	//定位状态更新
	//定位完成状态
	IF (iPosId<>-1) AND (bPosDone1 OR bPosDone2) THEN									                                             
	 		bGo_OK := TRUE;
			stAxis.Pos.State.bGo_Moving:=FALSE;		
			iPosId:=-1;
	END_IF;
	//定位完成与位置共同判断	 
	IF	 bRelEx THEN			 
		stAxis.Pos.State.bGo_OK	:=  bGo_OK (*AND (ABS((rPosEx + rRelStartPos)- stAxis.State.rActPos )<= stAxis.Parameter.rInPosValue)*);
	ELSE	
		stAxis.Pos.State.bGo_OK	:=  bGo_OK AND (ABS(stAxis.Pos.Par.rPos - stAxis.State.rActPos )<= stAxis.Parameter.rInPosValue);
	END_IF
		 
	//定位中状态
	IF (bPosBusy1 OR bPosBusy2)  THEN																						
	 	bGo_OK := FALSE;
		stAxis.Pos.State.bGo_Moving:=TRUE;				
	END_IF;
	//未定位中，清空定位ID号
	IF NOT bPosBusy1 AND NOT bPosBusy2 THEN  																
		iPosId:=-1;
	END_IF;
	
	//定位计时
	TonAxisMove(IN:=(iPosId <> -1), PT:= T#9999S);
	IF iPosId <> -1 THEN
		stAxis.Pos.State.rGo_CT:=TIME_TO_REAL(TonAxisMove.ET)/1000.0;	
	END_IF;	
END_IF;
{endregion}
END_ACTION

ACTION A_09_Stop:
{region "轴停止"}
IF TRUE THEN
	IF bHoming THEN
		lrStopMoveDec:=stAxis.Parameter.rStopDec * 1000.0;
	ELSE
		lrStopMoveDec:=stAxis.Parameter.rStopDec * 1000.0;
	END_IF;
		
	bStopMoveExe:= (stAxis.Control.bStop_M AND stSystem.bManual) OR stAxis.Control.bStop_A OR stSystem.bStop;
	IF bStopMoveExe (*AND NOT bStopMoveExeLast *)THEN
		bHomeJogBExe := FALSE ;
		bHomeJogFExe := FALSE ;	
		bHoming:= FALSE;
		iHomeStep:=0;
		iHomeStepPre := 0;
		stAxis.Pos.State.bGo_Moving:=FALSE;
		iPosId:=-1;
//		uiMotionCMD:=5;
	END_IF;
	bStopExe:= bHomeStop OR bStopMoveExe OR stAxis.State.bError OR stSystem.bEMG ;
	fbMcStop(
		Axis:= AxisRef, 
		Execute:= bStopExe  , 
		Deceleration:= lrStopMoveDec , 
		Jerk:= lrStopMoveDec * REAL#10.0	 , 
		Options:= , 
		Done=> , 
		Busy=> , 
		Active=> , 
		CommandAborted=> , 
		Error=> , 
		ErrorID=> );
	
	bHomeStop:=FALSE;
	IF stAxis.State.bStandStill AND ((stAxis.Control.bStop_M AND stSystem.bManual) OR stAxis.Control.bStop_A) THEN
		stAxis.Control.bStop_A:=FALSE;
		stAxis.Control.bStop_M:=FALSE;
	END_IF;
	bStopMoveExeLast:=bStopMoveExe;
END_IF;
{endregion}
END_ACTION

ACTION A_10_TrqCtr:
{region "力矩切换"}

// 转矩模式下，力矩切换
// 转矩6071目标转矩的单位为 0.1% ，上位机按照百分比输出，数据转换 *10

iTorqueTemp := REAL_TO_INT(stAxis.Parameter.rTorque *10)	;
	 
IF stAxis.State.siModeOfOperation = 10 THEN	// 驱动器处于转接模式时可设定力矩
	fbEcCoeSdoWriteExTargetTrq(
	sNetId:=strDriveAddressNetID , 
	nSlaveAddr:= uiDriveAddressSlaveAddr, 
	nSubIndex:= 16#00, 
	nIndex:= (16#6071 + (stAxis.Parameter.uiAxisChannelNum - 1)*16#800), 
	pSrcBuf:= ADR(iTorqueTemp), 
	cbBufLen:= SIZEOF(iTorqueTemp), 
	bExecute:= iTorqueTemp<> iTorqueTempOld , 
	tTimeout:= , 
	bCompleteAccess:= , 
	bBusy=> , 
	bError=> , 
	nErrId=> );	 
END_IF
iTorqueTempOld := iTorqueTemp;
	 
{endregion}
END_ACTION

ACTION A_11_StateOut:
{region "状态输出"}
//绝对值编码器电机在驱动器中设置好原点，默认原点OK
//增量式编码器需程序回零
IF  stAxis.Parameter.bAbsEnc AND stAxis.Control.bHome_A THEN
	stAxis.State.bHome_OK := TRUE;
	stAxis.Control.bHome_A:=FALSE;
ELSE
	stAxis.State.bHome_OK :=(AxisRef.Status.Homed OR stAxis.State.bHome_OK)
							AND NOT AxisRef.Status.DriveDeviceError;
	stAxis.State.bHoming :=(AxisRef.Status.Homing OR bHoming)
							AND NOT AxisRef.Status.DriveDeviceError;
END_IF;

//模轴和线性轴当前位置输出
stAxis.State.rActModuloPos := LREAL_TO_REAL(AxisRef.NcToPlc.ModuloActPos);
stAxis.State.rActPos := LREAL_TO_REAL(AxisRef.NcToPlc.ActPos);
//速度转矩加速度
stAxis.State.rActVel :=LREAL_TO_REAL(AxisRef.NcToPlc.ActVelo);
stAxis.State.rActTrq :=LREAL_TO_REAL(AxisRef.NcToPlc.ActTorque);
stAxis.State.rActAcc :=LREAL_TO_REAL(AxisRef.NcToPlc.ActAcc);
{endregion}
END_ACTION

ACTION A_12_Error:
{region "轴报警"}
//报警复位
IF ((stSystem.bReset OR stAxis.Control.bReset_A OR (stAxis.Control.bReset_M AND stSystem.bManual)) AND NOT bResetLast ) THEN
	FOR m:=1 TO 12 BY 1 DO
		stAxis.state.arErrorID[m]:= FALSE;
	END_FOR;
	stAxis.State.bWarning := FALSE;
	stAxis.State.bLightEror := FALSE;
	stAxis.State.bCriticalError :=FALSE;
END_IF;
bResetLast := stSystem.bReset;

//轴报警1-轴未使能
//屏蔽轴未使能报警
RtrigPowerOn(CLK:=stAxis.State.bPowerOK , Q=> );
//bHoming状态在驱动器回零时使用
IF NOT stAxis.State.bPowerOK AND NOT bHoming AND FALSE THEN
	stAxis.State.bLightEror := TRUE;
	stAxis.State.arErrorID[1]:=TRUE;
END_IF;
(*
IF RtrigPowerOn.Q THEN
	stAxis.State.bLightEror:=FALSE;
	stAxis.State.arErrorID[0]:=FALSE;
	stAxis.State.wstrErrorInfo:="--";
END_IF;
*)
	 
//轴报警2-轴NC报警
IF AxisRef.Status.ErrorID > 0 AND (NOT mcReset.Busy AND (NOT bHoming (*AND stAxis.Parameter.uiHomeMode <>6*))) THEN
	stAxis.State.bCriticalError := TRUE;
	stAxis.State.arErrorID[2]:=TRUE;
END_IF;
		  
//轴报警3-驱动器报警
TonReadDriveErrorCode(IN:=AxisRef.Status.DriveDeviceError,PT:=TIME#50MS);
IF AxisRef.Status.DriveDeviceError AND NOT mcReset.Busy AND TonReadDriveErrorCode.Q THEN
	stAxis.State.bCriticalError := TRUE;
	stAxis.State.arErrorID[3]:=TRUE;
END_IF;	 	 

//轴报警4-回零条件不满足报警
IF stAxis.Control.bHome_A AND NOT stAxis.Control.bHome_Con THEN
	stAxis.State.bLightEror := TRUE;
	stAxis.State.arErrorID[4]:=TRUE;
END_IF;	 

//轴报警5-正向JOG运行条件不满足报警
IF((stAxis.Control.bJogCw_A OR (stAxis.Control.bJogCw_M AND stSystem.bManual))AND NOT stAxis.Control.bJogCw_Con) THEN 
	stAxis.State.bLightEror := TRUE;
	stAxis.State.arErrorID[5]:=TRUE;
END_IF;

//轴报警6-负向JOG运行条件不满足报警
IF( (stAxis.Control.bJogCcw_A OR (stAxis.Control.bJogCcw_M AND stSystem.bManual)) AND NOT stAxis.Control.bJogCcw_Con) THEN 
	stAxis.State.bLightEror := TRUE;
	stAxis.State.arErrorID[6]:=TRUE;
END_IF;

//轴报警7-运行方向错误报警
IF ((stAxis.State.bPsw AND bHomeJogFExe) OR (stAxis.State.bNSw AND bHomeJogBExe)) AND NOT (stAxis.Parameter.uiHomeMode = 6 AND iHomeStepPre > 0 AND iHomeStep<1000) THEN
	bHomeJogFExe := FALSE;
	bHomeJogbExe := FALSE;
	bWrongDirection := TRUE;
END_IF;
IF stSystem.bReset OR stAxis.Control.bReset_A OR (stAxis.Control.bReset_M AND stSystem.bManual) THEN
	bWrongDirection := FALSE;
END_IF;
IF bWrongDirection THEN
	stAxis.State.bLightEror :=TRUE;
	stAxis.State.arErrorID[7]:=TRUE;
END_IF;
	 		   
//轴报警8-运行中碰正限位报警
RtrigJogB(CLK:=bJogBExe , Q=> );
IF (NOT stAxis.State.bPSw AND stAxis.State.bDirPositive ) AND NOT bHoming THEN 
	stAxis.State.bCriticalError :=TRUE;
	stAxis.State.arErrorID[8]:=TRUE;
END_IF;
IF RtrigJogB.Q AND stAxis.State.bPSw THEN
	stAxis.State.bCriticalError :=FALSE;
	stAxis.State.arErrorID[8]:=FALSE;
END_IF

// 轴报警9-运行中碰负限位报警
RtrigJogF(CLK:=bJogFExe , Q=> );
IF (NOT stAxis.State.bNSw AND stAxis.State.bDirNegative ) AND NOT bHoming THEN 
	stAxis.State.bCriticalError :=TRUE;
	stAxis.State.arErrorID[9]:=TRUE;
END_IF;
IF RtrigJogF.Q AND stAxis.State.bNSw THEN
	stAxis.State.bCriticalError :=FALSE;
	stAxis.State.arErrorID[9]:=FALSE;
END_IF

//
stAxis.state.bError := stAxis.State.bCriticalError OR stAxis.State.bLightEror ;
{endregion}


//报警输出	 
{region "SetAlarm"}
//SetAlarm
//轴报警从编号 101 开始, 12 个为一组
arrfbSetAlarm[1](
	bEnable:= TRUE, 
	iErrorID:= 100 + (UDINT_TO_INT(AxisREF.NcToPlc.AxisId)-1) * 12 + 1, 
	bExecute:= stAxis.State.arErrorID[1], 
	bReset:= stSystem.bReset OR stAxis.Control.bReset_A OR (stAxis.Control.bReset_M AND stSystem.bManual), 
	strErrorInfoEN:= 'not enabled', 
	wstrErrorInfoCN:= "轴未使能", 
	enumErrorClass:= 6, 
	 );
arrfbSetAlarm[2](
	bEnable:= TRUE, 
	iErrorID:= 100 + (UDINT_TO_INT(AxisREF.NcToPlc.AxisId)-1) * 12 + 2, 
	bExecute:= stAxis.State.arErrorID[2], 
	bReset:= stSystem.bReset OR stAxis.Control.bReset_A OR (stAxis.Control.bReset_M AND stSystem.bManual), 
	strErrorInfoEN:= 'NC alarm', 
	wstrErrorInfoCN:= "轴NC报警,报警代码-", 
	enumErrorClass:= 7,
	wstr1:=STRING_TO_WSTRING(stAxis.strName),
	D1:=UDINT_TO_DINT(AxisRef.Status.ErrorID),
	 );
arrfbSetAlarm[3](
	bEnable:= TRUE, 
	iErrorID:= 100+ (UDINT_TO_INT(AxisREF.NcToPlc.AxisId)-1) * 12 + 3, 
	bExecute:= stAxis.State.arErrorID[3], 
	bReset:= stSystem.bReset OR stAxis.Control.bReset_A OR (stAxis.Control.bReset_M AND stSystem.bManual), 
	strErrorInfoEN:= 'drive alarm', 
	wstrErrorInfoCN:= "驱动器报警,报警代码-", 
	enumErrorClass:= 7,
	wstr1:=STRING_TO_WSTRING(stAxis.strName),
	D1:=UDINT_TO_DINT(stAxis.State.uiDriveErrorCode),
	 );
arrfbSetAlarm[4](
	bEnable:= TRUE, 
	iErrorID:= 100+ (UDINT_TO_INT(AxisREF.NcToPlc.AxisId)-1) * 12 + 4, 
	bExecute:= stAxis.State.arErrorID[4], 
	bReset:= stSystem.bReset OR stAxis.Control.bReset_A OR (stAxis.Control.bReset_M AND stSystem.bManual), 
	strErrorInfoEN:= 'home condition not satisfied', 
	wstrErrorInfoCN:= "回零条件不满足", 
	wstr1:=STRING_TO_WSTRING(stAxis.strName),
	enumErrorClass:= 6, 
	 );	
arrfbSetAlarm[5](
	bEnable:= TRUE, 
	iErrorID:= 100+ (UDINT_TO_INT(AxisREF.NcToPlc.AxisId)-1) * 12 + 5, 
	bExecute:= stAxis.State.arErrorID[5], 
	bReset:= stSystem.bReset OR stAxis.Control.bReset_A OR (stAxis.Control.bReset_M AND stSystem.bManual), 
	strErrorInfoEN:= 'positive JOG condition not satisfied', 
	wstrErrorInfoCN:= "正向JOG运行条件不满足", 
	wstr1:=STRING_TO_WSTRING(stAxis.strName),
	enumErrorClass:= 6, 
	 );	 
arrfbSetAlarm[6](
	bEnable:= TRUE, 
	iErrorID:= 100+ (UDINT_TO_INT(AxisREF.NcToPlc.AxisId)-1) * 12 + 6, 
	bExecute:= stAxis.State.arErrorID[6], 
	bReset:= stSystem.bReset OR stAxis.Control.bReset_A OR (stAxis.Control.bReset_M AND stSystem.bManual), 
	strErrorInfoEN:= 'negative JOG condition not satisfied', 
	wstrErrorInfoCN:= "反向JOG运行条件不满足", 
	wstr1:=STRING_TO_WSTRING(stAxis.strName),
	enumErrorClass:= 6, 
	 );	 
arrfbSetAlarm[7](
	bEnable:= TRUE, 
	iErrorID:= 100+ (UDINT_TO_INT(AxisREF.NcToPlc.AxisId)-1) * 12 + 7, 
	bExecute:= stAxis.State.arErrorID[7], 
	bReset:= stSystem.bReset OR stAxis.Control.bReset_A OR (stAxis.Control.bReset_M AND stSystem.bManual), 
	strErrorInfoEN:= 'wrong direction of motion', 
	wstrErrorInfoCN:= "回零过程中JOG运行方向错误", 
	wstr1:=STRING_TO_WSTRING(stAxis.strName),
	enumErrorClass:= 6, 
	 );
arrfbSetAlarm[8](
	bEnable:= TRUE, 
	iErrorID:= 100+ (UDINT_TO_INT(AxisREF.NcToPlc.AxisId)-1) * 12 + 8, 
	bExecute:= stAxis.State.arErrorID[8], 
	bReset:= stSystem.bReset OR stAxis.Control.bReset_A OR (stAxis.Control.bReset_M AND stSystem.bManual), 
	strErrorInfoEN:= 'positive limit alarm', 
	wstrErrorInfoCN:=  "正限位报警", 
	wstr1:=STRING_TO_WSTRING(stAxis.strName),
	enumErrorClass:= 6, 
	 );
arrfbSetAlarm[9](
	bEnable:= TRUE, 
	iErrorID:= 100+ (UDINT_TO_INT(AxisREF.NcToPlc.AxisId)-1) * 12 + 9 , 
	bExecute:= stAxis.State.arErrorID[9], 
	bReset:= stSystem.bReset OR stAxis.Control.bReset_A OR (stAxis.Control.bReset_M AND stSystem.bManual), 
	strErrorInfoEN:= 'negative limit alarm', 
	wstrErrorInfoCN:=  "负限位报警",
	wstr1:=STRING_TO_WSTRING(stAxis.strName), 
	enumErrorClass:= 6, 
	 );		  
//轴报警10
arrfbSetAlarm[10](
	bEnable:= TRUE, 
	iErrorID:= 100+ (UDINT_TO_INT(AxisREF.NcToPlc.AxisId)-1) * 12 + 10, 
	bExecute:= stAxis.State.arErrorID[10], 
	bReset:= stSystem.bReset OR stAxis.Control.bReset_A OR (stAxis.Control.bReset_M AND stSystem.bManual), 
	strErrorInfoEN:= 'homing process interruption,step:', 
	wstrErrorInfoCN:=  "回零流程异常，步序-",	
	enumErrorClass:= 6, 
	wstr1:=STRING_TO_WSTRING(stAxis.strName),
	D1:=INT_TO_DINT(iHomeStep),
	 );

//轴报警11
arrfbSetAlarm[11](
	bEnable:= TRUE, 
	iErrorID:= 100 + (UDINT_TO_INT(AxisREF.NcToPlc.AxisId)-1) * 12 + 11, 
	bExecute:= stAxis.State.arErrorID[11], 
	bReset:= stSystem.bReset OR stAxis.Control.bReset_A OR (stAxis.Control.bReset_M AND stSystem.bManual), 
	strErrorInfoEN:= 'Positioning motion conditions are not met.', 
	wstrErrorInfoCN:=  "定位运动条件不满足", 
	wstr1:=STRING_TO_WSTRING(stAxis.strName),
	enumErrorClass:= 6, 
	 );
//轴报警12
arrfbSetAlarm[12](
	bEnable:= TRUE, 
	iErrorID:= 100 + (UDINT_TO_INT(AxisREF.NcToPlc.AxisId)-1) * 12 + 12, 
	bExecute:= stAxis.State.arErrorID[12], 
	bReset:= stSystem.bReset OR stAxis.Control.bReset_A OR (stAxis.Control.bReset_M AND stSystem.bManual), 
	strErrorInfoEN:= 'Positioning conditions not met during motion', 
	wstrErrorInfoCN:=  "运动中定位条件不满足", 
	wstr1:=STRING_TO_WSTRING(stAxis.strName),
	enumErrorClass:= 6, 
	 );
{endregion}
END_ACTION

END_FUNCTION_BLOCK

// ---- FB/61_Alarm/FB/FB_SetError.TcPOU
FUNCTION_BLOCK FB_SetError
VAR_INPUT
	//是否启用当前报警
    bEnable						:                   BOOL						;
	//当前报警的报警代码号
	iErrorID					:					INT							;
	//当前报警的触发信号输入
	bExecute						:					BOOL						;
END_VAR
VAR_INPUT
	//报警复位信号输入
	bReset						:					BOOL						;
	// 报警信息-英文字符
	strErrorInfoEN				: 					STRING						;
	// 报警信息-中文字符
	wstrErrorInfoCN				: 					WSTRING						;
	//当前报警的等级设定
	enumErrorClass				:					Enum_ErrorClass				;
END_VAR
VAR_INPUT
	//报警发生时，需要触发的动作，1-4中任意选择。                           						
	bAlarmAction1				:					BOOL						;
	bAlarmAction2				:					BOOL						;
	bAlarmAction3				:					BOOL						;
	bAlarmAction4				:					BOOL						;
	// 报警代码的对应轴名称，驱动器报警时可以调用
	wstr1						: 					WSTRING						;
	// 报警代码，NC报警代码，驱动器报警代码
	D1							:					DINT						;
END_VAR
VAR_OUTPUT
	// 报警启用标志位
	bEnabled					: 					BOOL						;
	// 报警发生标志位
	bErrorOccur					:					BOOL						;
END_VAR
VAR
	(**暂时不启用，需要时添加至输入变量中**)
	//是否对当前报警启用滤波功能(**暂时不启用，需要时添加至输入变量中**)
   bFilterOn					:                  	BOOL:=FALSE					;
	//滤波功能的时间设定(**暂时不启用，需要时添加至输入变量中**)
   timeFilter					:                   TIME := TIME#0MS			;	
	// 是否使用reset信号复位:  true=复位信号为1时且触发信号为0时，复位报警状态;  false=触发信号为0时自动复位报警信号(**暂时不启用，需要时添加至输入变量中**)
	bResetSignalUse				:					BOOL := TRUE				;	
	//设定是否将当前报警记录到历史记录中(**暂时不启用，需要时添加至输入变量中**)
   	bSavetoHistory				:                 	BOOL := TRUE				;
	strVersion: STRING;

	
	// 获取报警时间
	rtrigGetTime				:          			R_TRIG						;
  	// 滤波延时
	tonFilter					:               	TON							;	
 	// 报警复位信号下降沿
	ftrigResetExe				:          			F_TRIG						;	
	i							:                 	INT							;
	strTemp						: 					STRING						;
	fbFormatStringDateTime		: 					FB_FormatString				;
	strDateTime					: 					STRING(255)					;
	wstrErrorMessage			: 					WSTRING						;
	bFirstRun: BOOL := true;
	ton100msDelay: TON;
END_VAR

(***
by Yu
	
	2025-07-23	报警设置功能块，每一个报警都需实例化一次。
	2025-07-24	输出的报警信息中不同时整合报警时间和报警ID号,减少字符的使用长度。报警时间、报警ID号、报警信息，以结构体的形式分别输出。
	2025-10-29	报警发生时，增加获取系统时间判定，防止出现开机一瞬间，系统时间还未获取时，出现的错误时间报警


***)
//当前版本更新时间
strVersion := '2025-10-29' ;

//初始化
IF bFirstRun THEN
;
END_IF


//报警ID号超范围直接退出
IF iErrorID> iErrorIDMax OR iErrorID< 1 THEN
	RETURN;
END_IF

//报警复位
 ftrigResetExe(CLK:=bReset);
 IF ((bResetSignalUse AND  ftrigResetExe.Q)OR NOT bResetSignalUse )AND NOT bExecute OR NOT bEnable THEN
    bErrorOccur:=FALSE;
    arrstError[iErrorID].bAlarmAction1:=FALSE;
    arrstError[iErrorID].bAlarmAction2:=FALSE;
    arrstError[iErrorID].bAlarmAction3:=FALSE;
    arrstError[iErrorID].bAlarmAction4:=FALSE;
	arrstError[iErrorID].bEnabled:=bEnable;
	arrstError[iErrorID].bErrorOccur:=bErrorOccur;
	arrstError[iErrorID].bErrorExe:=bExecute;
	arrstError[iErrorID].enumErrorClass:=enumErrorClass;
	arrstError[iErrorID].iErrorID:=iErrorID;
	arrstError[iErrorID].bResetExe:=bReset;
	arrstError[iErrorID].bResetSignalUse:=bResetSignalUse;
 END_IF
 
	
//滤波延时
tonFilter(IN:=bFilterOn AND bExecute , PT:=timeFilter );

//报警发生上升沿触发且系统时间读取成功
rtrigGetTime(CLK:=((NOT bFilterOn ) OR (bFilterOn AND tonFilter.Q))AND bEnable AND bExecute AND bGetSystemTimeDone  );

//将当前系统时间写入到对应的轴结构体中 
IF rtrigGetTime.Q THEN
	arrstError[iErrorID].dtErrorOccorTime:=SYSTEMTIME_TO_DT(tActSystemTime);
END_IF

//报警发生时触发
IF ((NOT bFilterOn ) OR (bFilterOn AND tonFilter.Q)) AND bEnable AND bExecute AND bGetSystemTimeDone THEN
	//报警发生标志位
	bErrorOccur:=TRUE;
	//将报警后的触发动作写入对应的ErrorID号下
	arrstError[iErrorID].bAlarmAction1:=bAlarmAction1;
	arrstError[iErrorID].bAlarmAction2:=bAlarmAction2;
	arrstError[iErrorID].bAlarmAction3:=bAlarmAction3;
	arrstError[iErrorID].bAlarmAction4:=bAlarmAction4;
	//设定此ErrorID号报警是否启用
	arrstError[iErrorID].bEnabled:=bEnable;
	//此ErrorID号报警发生标志位
	arrstError[iErrorID].bErrorOccur:=bErrorOccur;
	//此ErrorID号报警触发信号
	arrstError[iErrorID].bErrorExe:=bExecute;
	//此ErrorID号报警警报等级	
	arrstError[iErrorID].enumErrorClass:=enumErrorClass;
	//此ErrorID号报警报警ID	
	arrstError[iErrorID].iErrorID:=iErrorID;
	//此ErrorID号报警报警复位信号		
	arrstError[iErrorID].bResetExe:=bReset;
	//设定此ErrorID号报警是否与复位信号联动
	arrstError[iErrorID].bResetSignalUse:=bResetSignalUse;
END_IF

//报警发生时的时间转换程string类型。时间-报警ID号-报警信息，组合输出
IF rtrigGetTime.Q THEN
	fbFormatStringDateTime(
		sFormat:= '%D-%D-%D-%D:%D:%D',
		arg1:= F_WORD(tActSystemTime.wYear),
		arg2:= F_WORD(tActSystemTime.wMonth),
		arg3:= F_WORD(tActSystemTime.wDay),
		arg4:= F_WORD(tActSystemTime.wHour),
		arg5:= F_WORD(tActSystemTime.wMinute),
		arg6:= F_WORD(tActSystemTime.wSecond),
		sOut=> strDateTime
		);
	//默认使用中文报警信息
	IF bLanguageSet=1 THEN
		wstrErrorMessage:=STRING_TO_WSTRING(strErrorInfoEN);
	ELSE
		wstrErrorMessage:=wstrErrorInfoCN;
	END_IF	
	F_FormatWstringErrInfo(wstrIn:=wstrErrorMessage,wstrPreMessage:=wstr1,diMessage:=D1,wstrOut=>wstrErrorMessage);	
	//整合需要添加的字符后，直接输出，不添加报警时间以及报警ID，减少字符的长度
	arrstError[iErrorID].wstrErrorMessage := wstrErrorMessage ;	
//	wstrErrorMessage:=	WCONCAT(WCONCAT(WCONCAT("ID",INT_TO_WSTRING(iErrorID)),","),wstrErrorMessage);		
//	arrstError[iErrorID].wstrErrorMessage := WCONCAT(WCONCAT(STRING_TO_WSTRING(strDateTime),"-"),wstrErrorMessage);	
END_IF
	   

//当选择将此报警记录如历史报警记录后，触发记录。最大记录数组200组。数据向后依次排列
IF bSavetoHistory  AND rtrigGetTime.Q THEN
	iHistoryErrorNum:=iHistoryErrorNum+1;
	IF iHistoryErrorNum>=200 THEN
		iHistoryErrorNum:=200;
	END_IF
	IF iHistoryErrorNum>=2 THEN
		FOR i:=iHistoryErrorNum TO 2 BY -1 DO
			arrstHistoryError[i]:=arrstHistoryError[i-1];
		END_FOR
	END_IF
 	arrstHistoryError[1].iErrorID:=iErrorID;
	arrstHistoryError[1].dtErrorTime:=arrstError[iErrorID].dtErrorOccorTime;
  	arrstHistoryError[1].wstrErrorMessage:=arrstError[iErrorID].wstrErrorMessage;
END_IF

END_FUNCTION_BLOCK

// ---- FB/61_Alarm/FB/F_FormatWstringErrInfo.TcPOU
FUNCTION F_FormatWstringErrInfo : WSTRING
FUNCTION F_FormatWstringErrInfo : BOOL
VAR_INPUT
	wstrIn:			WSTRING;
	// 前缀
	wstrPreMessage: WSTRING;
	// 后缀
	diMessage:					DINT;
END_VAR
VAR_OUTPUT
	wstrOut:			WSTRING;
END_VAR
VAR
	strVersion: STRING;
	iVar0: INT;
	iVar1: INT;
	iVar2: DINT;
	wstrTemp: WSTRING;
END_VAR

(***
by Yu
	
	2025-07-23	实现对信息的组合,前缀为 WSTRING 变量，后缀添加 DINT 型变量。可用于添加 轴名称-报警信息-报警代码 。

***)
//当前版本更新时间
strVersion := '2025-07-23' ;

//
iVar0:=WLEN(wstrIn);
iVar1:=WLEN(wstrPreMessage);
iVar2:=diMessage;

IF iVar1 <>0 AND iVar2 <>0 THEN
	wstrTemp := WCONCAT(wstrPreMessage,wstrIn);
	wstrOut := WCONCAT(wstrtemp,DINT_TO_WSTRING(diMessage));
ELSIF iVar1 = 0 AND iVar2 <> 0  THEN
	wstrOut := WCONCAT(wstrIn,DINT_TO_WSTRING(diMessage));
ELSIF iVar1 <>0 AND iVar2 =0 THEN
	wstrOut := WCONCAT(wstrPreMessage,wstrIn);	
ELSE
	wstrOut := wstrIn;
END_IF

END_FUNCTION

// ---- FB/01_Axis/FB/FB_TouchProbe_Home_Bylimit.TcPOU
FUNCTION_BLOCK FB_TouchProbe_Home_Bylimit
VAR_INPUT	
		bCMD_HomeExecute			:REFERENCE TO BOOL;			(* 执行回零*)
		bCMD_Reset					:REFERENCE TO BOOL;			(* 回零错误复位*)
		bCMD_EnableState			:BOOL;						(* 使能状态输入*)	
		bCMD_StartHomeIndex			:BOOL;						(* 是否使用索引回零*)
		eCMD_HomeDirection			:MC_Direction;				(* 回原点方向*)
		bCMD_PositiveLimit			:BOOL;						(* 正限位传感器*)
		bCMD_NegativeLimit			:BOOL;						(* 负限位传感器*)
		rCMD_HomePosition			:LREAL;						(* 设定回原点位置*)
		rCMD_TowardsVelSetValue		:LREAL;						(* 靠近原点速度*)
		rCMD_OffVelSetValue			:LREAL;						(* 离开原点速度*)
	    stHomeAdsGroup				:ST_HomeAdsGroup;			(* ADS地址信息*)

END_VAR
VAR_OUTPUT
		bResult_HomeDone			:BOOL;						(* 回原点完成状态*)
		bResult_HomeBusy			:BOOL;						(* 正在回原点中状态*)
		bResult_HomeError			:BOOL;						(* 回原点错误状态*)
		nResult_HomeErrorID			:UDINT;						(* 回原点错误代码*)
END_VAR
VAR_IN_OUT
		axis						:AXIS_REF;
END_VAR
VAR
	  
		mcHome						:MC_Home;
		mcReset						:MC_Reset;
		fbReadParameter				:ARRAY [0..4] OF ADSREAD;
		fbwriteParameter			:ARRAY [0..4] OF ADSWRITE;
		rTowardsVelActValue			:LREAL;		
		rOffVelActValue				:LREAL;
		nHomeSenorSetValue			:INT;
		nHomeSensorActValue			:INT;
		nHomeSynSetValue			:WORD;
		nHomeSynActValue			:WORD;
		nHomeSetRefMode				:DINT;
		nHomeActRefMode				:DINT;
		mcHomeStatus				:ST_McOutputs;
		fbReadParaStatus			:ARRAY [0..4] OF ST_McOutputs;
		fbWriteParaStatus			:ARRAY [0..4] OF ST_McOutputs;
		posEdge_bCMD_HomeExecute	:R_TRIG;
		posEdge_bCMD_Reset			:R_TRIG;
		negEdge_bCMD_Calibration	:F_TRIG;
		ton_bCMD_HomeExecute		:TON;
		ton_nStep					:TON;
		ton_bCMD_Reset				:TON;
		ton_McReset					:TON;
		ton_HomErr                  :TON;
		nStep						:E_HomeStep;
		mcMoveAbs					:MC_MoveAbsolute;
END_VAR

posEdge_bCMD_HomeExecute(CLK:=bCMD_HomeExecute AND bCMD_EnableState AND NOT bResult_HomeError AND NOT bResult_HomeBusy);
ton_bCMD_HomeExecute(IN:=bCMD_HomeExecute,PT:=T#100MS);

IF posEdge_bCMD_HomeExecute.Q  THEN
	nStep:=AckHomeDirection;
ELSIF	ton_bCMD_HomeExecute.Q THEN
	 bCMD_HomeExecute:=FALSE;
END_IF


IF eCMD_HomeDirection=MC_Direction.MC_Positive_Direction  THEN
	mcHome.bCalibrationCam:=bCMD_PositiveLimit;
ELSIF eCMD_HomeDirection=MC_Direction.MC_Negative_Direction THEN
		mcHome.bCalibrationCam:=bCMD_NegativeLimit;
END_IF

CASE nStep OF
IndexHomeInital:
	ton_nStep(IN:=FALSE);		
	bResult_HomeBusy:=FALSE;
	mcHome.Execute:=FALSE;
	mcMoveAbs.Execute:=FALSE;
	fbReadParameter[0].READ:=fbReadParameter[1].READ:=fbReadParameter[2].READ:=fbReadParameter[3].READ:=fbReadParameter[4].READ:=FALSE;
	fbwriteParameter[0].WRITE:=fbwriteParameter[1].WRITE:=fbwriteParameter[2].WRITE:=fbwriteParameter[3].WRITE:=fbwriteParameter[4].WRITE:=FALSE;
	IF axis.Status.Error OR mcHome.Error THEN
		nStep:=IndexHomeErrorState;
	END_IF
AckHomeDirection:
	bResult_HomeBusy:=TRUE;
	bResult_HomeDone:=FALSE;
	IF bCMD_StartHomeIndex THEN
		nHomeSetRefMode:=2;
	ELSE
		nHomeSetRefMode:=0;  
	END_IF
	IF eCMD_HomeDirection=MC_Direction.MC_Positive_Direction   THEN
		nHomeSenorSetValue:=0;
		nHomeSynSetValue:=1;
		nStep:=SetParameter;
	ELSIF eCMD_HomeDirection=MC_Direction.MC_Negative_Direction THEN
		nHomeSenorSetValue:=1;
		nHomeSynSetValue:=0;
		nStep:=SetParameter;
	ELSE
		nStep:=IndexHomeErrorState;
	END_IF
SetParameter:
	fbwriteParameter[0].WRITE:=fbwriteParameter[1].WRITE:=fbwriteParameter[2].WRITE:=
	fbwriteParameter[3].WRITE:=fbwriteParameter[4].WRITE:=TRUE;
	nStep:=SetParameterState;	
SetParameterState:
	ton_nStep(IN:=TRUE,PT:=T#100MS);
	IF ton_nStep.Q AND NOT fbWriteParaStatus[0].Busy AND NOT fbWriteParaStatus[1].Busy AND NOT fbWriteParaStatus[2].Busy AND 
		NOT fbWriteParaStatus[3].BUSY AND NOT fbWriteParaStatus[4].BUSY  THEN
		nStep:=ReadParameter;
		fbwriteParameter[0].WRITE:=fbwriteParameter[1].WRITE:=fbwriteParameter[2].WRITE
		:=fbwriteParameter[3].WRITE:=fbwriteParameter[4].WRITE:=FALSE;
	ELSIF ton_nStep.Q AND (fbWriteParaStatus[0].Error OR fbWriteParaStatus[1].Error OR fbWriteParaStatus[2].Error OR
		fbWriteParaStatus[3].Error OR fbWriteParaStatus[4].Error) THEN
		nStep:=IndexHomeErrorState;
	END_IF
ReadParameter:
	fbReadParameter[0].READ:=fbReadParameter[1].READ:=fbReadParameter[2].READ:=
	fbReadParameter[3].READ:=fbReadParameter[4].READ:=TRUE;
	nStep:=ReadParameterState;
ReadParameterState:
	ton_nStep(IN:=TRUE,PT:=T#100MS);
	
	IF ton_nStep.Q AND NOT fbReadParaStatus[0].BUSY AND NOT fbReadParaStatus[1].BUSY AND NOT fbReadParaStatus[2].BUSY
		AND NOT fbReadParaStatus[3].BUSY AND NOT fbReadParaStatus[4].BUSY THEN
		fbReadParameter[0].READ:=fbReadParameter[1].READ:=fbReadParameter[2].READ:=
		fbReadParameter[3].READ:=fbReadParameter[4].READ:=FALSE;
		nStep:=AckParameter;
	ELSIF ton_nStep.Q AND (fbReadParaStatus[0].Error OR fbReadParaStatus[1].Error OR fbReadParaStatus[2].Error OR 
		fbReadParaStatus[3].Error OR fbReadParaStatus[4].Error) THEN
		nStep:=IndexHomeErrorState;
	END_IF
AckParameter:
	IF rTowardsVelActValue=rCMD_TowardsVelSetValue AND rOffVelActValue=rCMD_OffVelSetValue AND
		nHomeSensorActValue=nHomeSenorSetValue AND nHomeSynActValue=nHomeSynSetValue 
		AND nHomeActRefMode=nHomeSetRefMode  THEN
		nStep:=ExecuteToOrigin;
	ELSE
		nStep:=IndexHomeErrorState;
	END_IF
ExecuteToOrigin:
	mcHome.Execute:=TRUE;
	nStep:=HomeMonitorState;
HomeMonitorState:
	IF mcHome.Done THEN
		mcHome.Execute:=FALSE;
		nStep:=HomeMoveABS;
	ELSIF mcHome.Error OR axis.Status.Error THEN
		nStep:=IndexHomeErrorState;
	END_IF	
	IF eCMD_HomeDirection=MC_Direction.MC_Positive_Direction AND bCMD_NegativeLimit AND ton_HomErr.Q THEN
		mcReset.Execute:=TRUE;
		nStep:=IndexHomeErrorState;
	ELSIF eCMD_HomeDirection=MC_Direction.MC_Negative_Direction AND bCMD_PositiveLimit AND ton_HomErr.Q THEN
		mcReset.Execute:=TRUE;
		nStep:=IndexHomeErrorState;
	END_IF
HomeMoveABS:
	mcMoveAbs.Execute:=TRUE;	
	IF mcMoveAbs.Done THEN
		mcMoveAbs.Execute:=FALSE;
		nStep:=ExecuteHomeDone;
	ELSIF axis.Status.Error OR mcMoveAbs.Error THEN
		nStep:=IndexHomeErrorState;
	END_IF
ExecuteHomeDone:
	bResult_HomeBusy:=FALSE;
	bResult_HomeDone:=TRUE;
	nStep:=E_HomeStep.IndexHomeInital;
IndexHomeErrorState:
	bResult_HomeBusy:=FALSE;
	bResult_HomeDone:=FALSE;
	bResult_HomeError:=TRUE;
	mcHome.Execute:=FALSE;
	mcMoveAbs.Execute:=FALSE;
	nStep:=IndexHomeInital;
END_CASE
// 超时定时器
ton_HomErr(IN:=bResult_HomeBusy , PT:=T#20S , Q=> , ET=> );

ACT_AxisControl();
ACT_ErrorID();
ACT_Reset();

ACTION ACT_AxisControl:
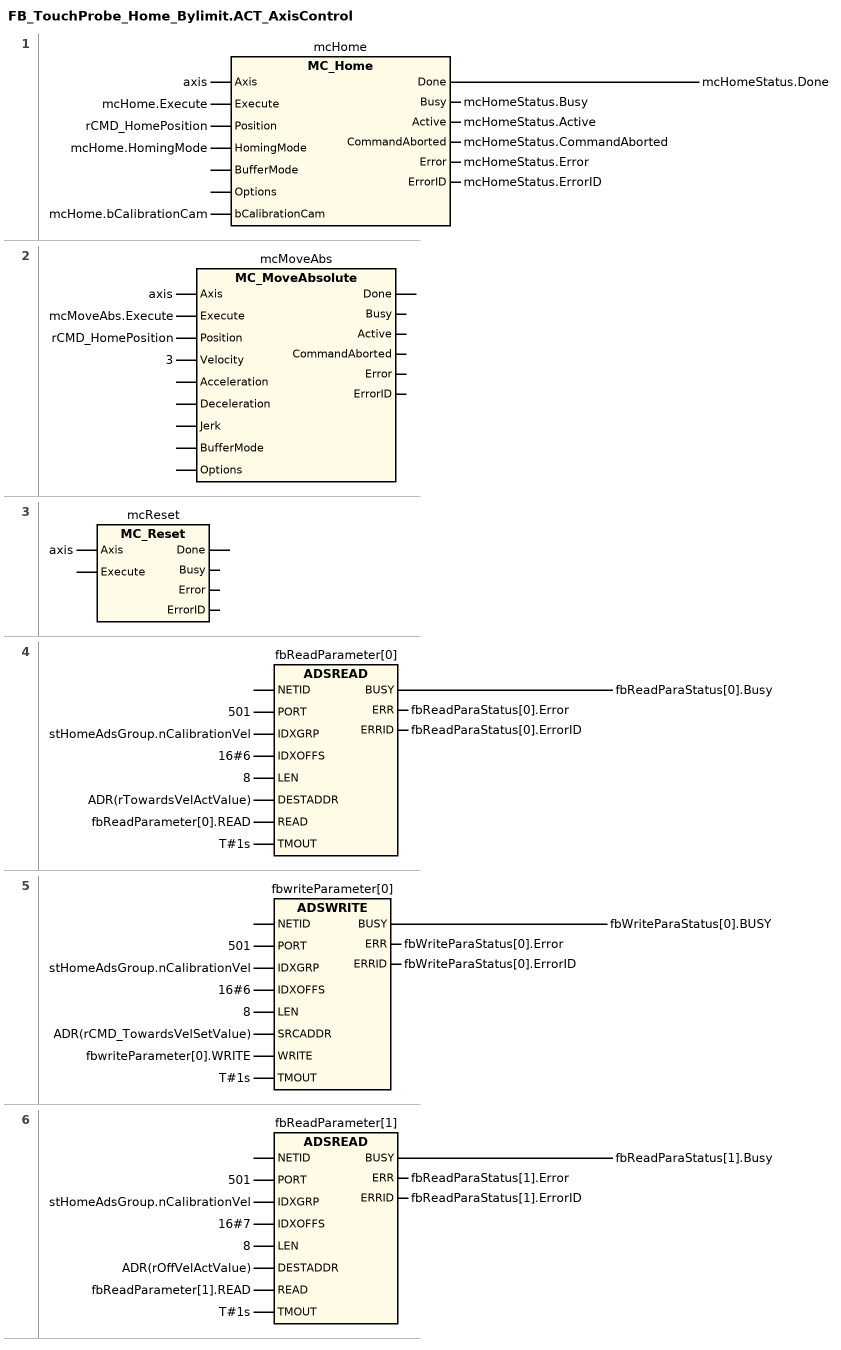
// NETWORK 1
mcHome(
    Axis := axis,
    Execute := mcHome.Execute,
    Position := rCMD_HomePosition,
    HomingMode := mcHome.HomingMode,
    bCalibrationCam := mcHome.bCalibrationCam,
    Busy => mcHomeStatus.Busy,
    Active => mcHomeStatus.Active,
    CommandAborted => mcHomeStatus.CommandAborted,
    Error => mcHomeStatus.Error,
    ErrorID => mcHomeStatus.ErrorID); // MC_Home
mcHomeStatus.Done := mcHome.Done;

// NETWORK 2
mcMoveAbs(Axis := axis, Execute := mcMoveAbs.Execute, Position := rCMD_HomePosition, Velocity := 3); // MC_MoveAbsolute

// NETWORK 3
mcReset(Axis := axis); // MC_Reset

// NETWORK 4
fbReadParameter[0](
    PORT := 501,
    IDXGRP := stHomeAdsGroup.nCalibrationVel,
    IDXOFFS := 16#6,
    LEN := 8,
    DESTADDR := ADR(rTowardsVelActValue),
    READ := fbReadParameter[0].READ,
    TMOUT := T#1s,
    ERR => fbReadParaStatus[0].Error,
    ERRID => fbReadParaStatus[0].ErrorID); // ADSREAD
fbReadParaStatus[0].Busy := fbReadParameter[0].BUSY;

// NETWORK 5
fbwriteParameter[0](
    PORT := 501,
    IDXGRP := stHomeAdsGroup.nCalibrationVel,
    IDXOFFS := 16#6,
    LEN := 8,
    SRCADDR := ADR(rCMD_TowardsVelSetValue),
    WRITE := fbwriteParameter[0].WRITE,
    TMOUT := T#1s,
    ERR => fbWriteParaStatus[0].Error,
    ERRID => fbWriteParaStatus[0].ErrorID); // ADSWRITE
fbWriteParaStatus[0].BUSY := fbwriteParameter[0].BUSY;

// NETWORK 6
fbReadParameter[1](
    PORT := 501,
    IDXGRP := stHomeAdsGroup.nCalibrationVel,
    IDXOFFS := 16#7,
    LEN := 8,
    DESTADDR := ADR(rOffVelActValue),
    READ := fbReadParameter[1].READ,
    TMOUT := T#1s,
    ERR => fbReadParaStatus[1].Error,
    ERRID => fbReadParaStatus[1].ErrorID); // ADSREAD
fbReadParaStatus[1].Busy := fbReadParameter[1].BUSY;

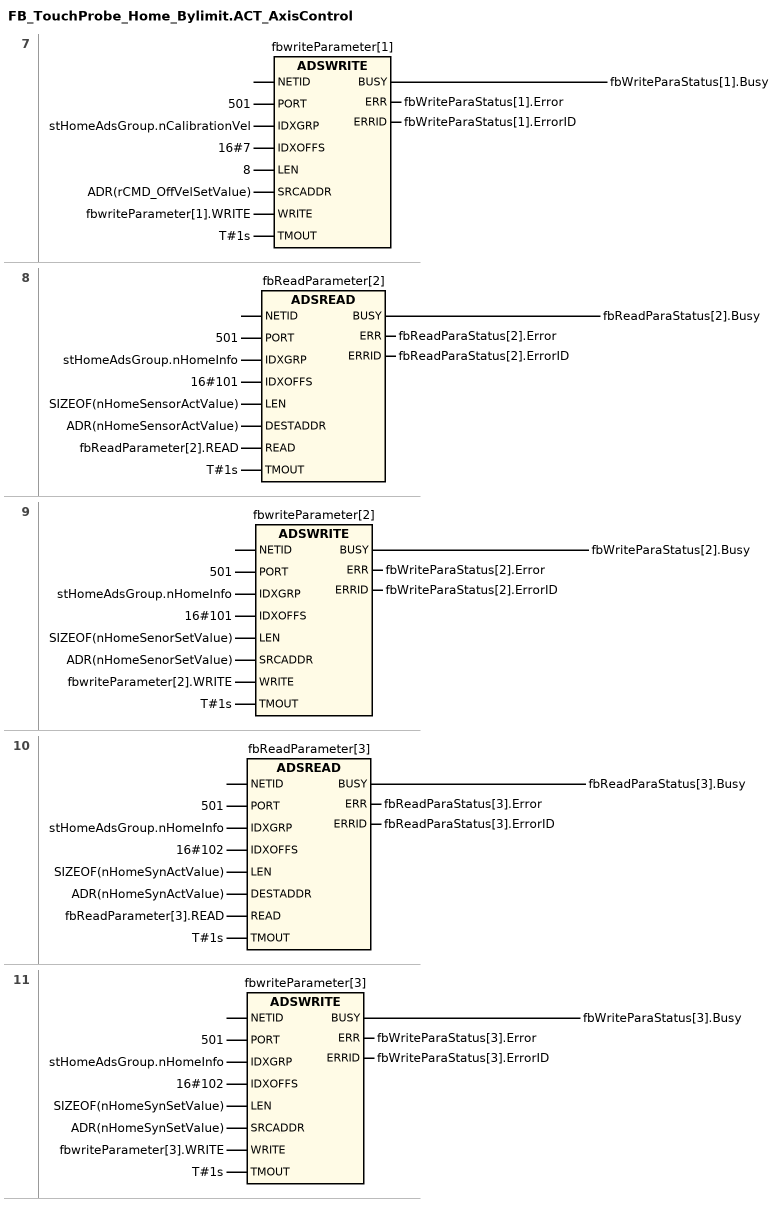
// NETWORK 7
fbwriteParameter[1](
    PORT := 501,
    IDXGRP := stHomeAdsGroup.nCalibrationVel,
    IDXOFFS := 16#7,
    LEN := 8,
    SRCADDR := ADR(rCMD_OffVelSetValue),
    WRITE := fbwriteParameter[1].WRITE,
    TMOUT := T#1s,
    ERR => fbWriteParaStatus[1].Error,
    ERRID => fbWriteParaStatus[1].ErrorID); // ADSWRITE
fbWriteParaStatus[1].Busy := fbwriteParameter[1].BUSY;

// NETWORK 8
fbReadParameter[2](
    PORT := 501,
    IDXGRP := stHomeAdsGroup.nHomeInfo,
    IDXOFFS := 16#101,
    LEN := SIZEOF(nHomeSensorActValue),
    DESTADDR := ADR(nHomeSensorActValue),
    READ := fbReadParameter[2].READ,
    TMOUT := T#1s,
    ERR => fbReadParaStatus[2].Error,
    ERRID => fbReadParaStatus[2].ErrorID); // ADSREAD
fbReadParaStatus[2].Busy := fbReadParameter[2].BUSY;

// NETWORK 9
fbwriteParameter[2](
    PORT := 501,
    IDXGRP := stHomeAdsGroup.nHomeInfo,
    IDXOFFS := 16#101,
    LEN := SIZEOF(nHomeSenorSetValue),
    SRCADDR := ADR(nHomeSenorSetValue),
    WRITE := fbwriteParameter[2].WRITE,
    TMOUT := T#1s,
    ERR => fbWriteParaStatus[2].Error,
    ERRID => fbWriteParaStatus[2].ErrorID); // ADSWRITE
fbWriteParaStatus[2].Busy := fbwriteParameter[2].BUSY;

// NETWORK 10
fbReadParameter[3](
    PORT := 501,
    IDXGRP := stHomeAdsGroup.nHomeInfo,
    IDXOFFS := 16#102,
    LEN := SIZEOF(nHomeSynActValue),
    DESTADDR := ADR(nHomeSynActValue),
    READ := fbReadParameter[3].READ,
    TMOUT := T#1s,
    ERR => fbReadParaStatus[3].Error,
    ERRID => fbReadParaStatus[3].ErrorID); // ADSREAD
fbReadParaStatus[3].Busy := fbReadParameter[3].BUSY;

// NETWORK 11
fbwriteParameter[3](
    PORT := 501,
    IDXGRP := stHomeAdsGroup.nHomeInfo,
    IDXOFFS := 16#102,
    LEN := SIZEOF(nHomeSynSetValue),
    SRCADDR := ADR(nHomeSynSetValue),
    WRITE := fbwriteParameter[3].WRITE,
    TMOUT := T#1s,
    ERR => fbWriteParaStatus[3].Error,
    ERRID => fbWriteParaStatus[3].ErrorID); // ADSWRITE
fbWriteParaStatus[3].Busy := fbwriteParameter[3].BUSY;

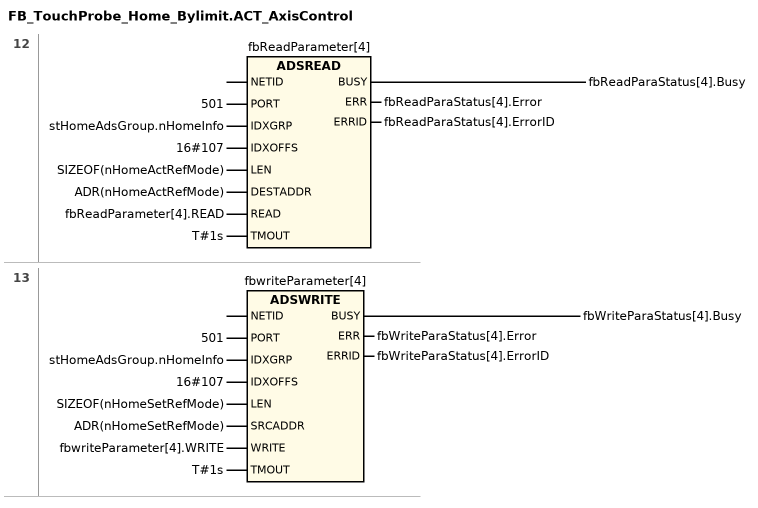
// NETWORK 12
fbReadParameter[4](
    PORT := 501,
    IDXGRP := stHomeAdsGroup.nHomeInfo,
    IDXOFFS := 16#107,
    LEN := SIZEOF(nHomeActRefMode),
    DESTADDR := ADR(nHomeActRefMode),
    READ := fbReadParameter[4].READ,
    TMOUT := T#1s,
    ERR => fbReadParaStatus[4].Error,
    ERRID => fbReadParaStatus[4].ErrorID); // ADSREAD
fbReadParaStatus[4].Busy := fbReadParameter[4].BUSY;

// NETWORK 13
fbwriteParameter[4](
    PORT := 501,
    IDXGRP := stHomeAdsGroup.nHomeInfo,
    IDXOFFS := 16#107,
    LEN := SIZEOF(nHomeSetRefMode),
    SRCADDR := ADR(nHomeSetRefMode),
    WRITE := fbwriteParameter[4].WRITE,
    TMOUT := T#1s,
    ERR => fbWriteParaStatus[4].Error,
    ERRID => fbWriteParaStatus[4].ErrorID); // ADSWRITE
fbWriteParaStatus[4].Busy := fbwriteParameter[4].BUSY;
END_ACTION

ACTION ACT_ErrorID:
nResult_HomeErrorID:=mcHome.ErrorID;
END_ACTION

ACTION ACT_Reset:
posEdge_bCMD_Reset(CLK:=bCMD_Reset);
ton_bCMD_Reset(IN:=bCMD_Reset,PT:=T#100MS);
ton_McReset(IN:=mcReset.Execute,PT:=T#100MS);
IF posEdge_bCMD_Reset.Q THEN
	bResult_HomeBusy:=FALSE;
	bResult_HomeDone:=FALSE;
	bResult_HomeError:=FALSE;
	nStep:=IndexHomeInital;
	mcReset.Execute:=TRUE;
	mcMoveAbs.Execute:=FALSE;
ELSIF ton_bCMD_Reset.Q THEN
	bCMD_Reset:=FALSE;
END_IF

IF ton_McReset.Q THEN
	mcReset.Execute:=FALSE;
END_IF
END_ACTION

END_FUNCTION_BLOCK

// ---- FB/01_Axis/FB/FB_Drive_Home.TcPOU
FUNCTION_BLOCK FB_Drive_Home
VAR_INPUT	
		bCMD_EnableState			:BOOL;						(* 使能状态输入*)	
		bCMD_siHomeMethod			:SINT;						(* 驱动器回圆方法*)
		bCMD_PositiveLimit			:BOOL;						(* 正限位传感器*)
		bCMD_NegativeLimit			:BOOL;						(* 负限位传感器*)
		rCMD_HomePosition			:LREAL;						(* 设定回原点位置*)
		rCMD_TowardsVelSetValue		:LREAL;						(* 靠近原点速度*)
		rCMD_OffVelSetValue			:LREAL;						(* 离开原点速度*)	
        bCMD_HomeExecute			:REFERENCE TO BOOL;			(* 执行回零*)
		bCMD_Reset					:REFERENCE TO BOOL;			(* 回零错误复位*)	
		stHomeCoEGroup				:ST_HomeCoEGroup;			(* coe信息*)
END_VAR
VAR_OUTPUT
	    bProcessPowerCtrl           :BOOL;
		bResult_HomeDone			:BOOL;						(* 回原点完成状态*)
		bResult_HomeBusy			:BOOL;						(* 正在回原点中状态*)
		bResult_HomeError			:BOOL;						(* 回原点错误状态*)
		nResult_HomeErrorID			:UDINT;						(* 回原点错误代码*)
END_VAR
VAR_IN_OUT
		axis						:AXIS_REF;
END_VAR
VAR
		mcHome						:MC_Home;
		mcReset						:MC_Reset;
		mcjog                       :MC_Jog;	
		mcMoveAbs					:MC_MoveAbsolute;
        FB_EcCoESdoWrite_6098:    FB_EcCoESdoWrite;
	    FB_EcCoESdoWrite_6099_01: FB_EcCoESdoWrite;
	    FB_EcCoESdoWrite_6099_02: FB_EcCoESdoWrite;
	    FB_EcCoESdoWrite_609A:    FB_EcCoESdoWrite;
	    FB_EcCoESdoWrite_607C:    FB_EcCoESdoWrite;
		uiStatusWord: UINT;
	    FB_EcCoESdoRead_6041: FB_EcCoESdoRead;
		fbReadParameter				:ARRAY [0..4] OF ADSREAD;
		fbwriteParameter			:ARRAY [0..4] OF ADSWRITE;
		rTowardsVelActValue			:LREAL;		
		rOffVelActValue				:LREAL;
		nHomeSenorSetValue			:INT;
		nHomeSensorActValue			:INT;
		nHomeSynSetValue			:WORD;
		nHomeSynActValue			:WORD;
		nHomeSetRefMode				:DINT;
		nHomeActRefMode				:DINT;
		mcHomeStatus				:ST_McOutputs;
		fbReadParaStatus			:ARRAY [0..4] OF ST_McOutputs;
		fbWriteParaStatus			:ARRAY [0..4] OF ST_McOutputs;
		posEdge_bCMD_HomeExecute	:R_TRIG;
		posEdge_bCMD_Reset			:R_TRIG;
		negEdge_bCMD_Calibration	:F_TRIG;
		ton_bCMD_HomeExecute		:TON;
		ton_nStep					:TON;
		ton_bCMD_Reset				:TON;
		ton_McReset					:TON;
		ton_HomErr                  :TON;
		nStep						:INT;
		
		
		fbEcCoESdoReadErrCode: FB_EcCoESdoRead                      ;           // 读COE 力矩
	    fbEcCoESdoWriteHMethod: FB_EcCoESdoWrite                  ;           // 写COE 回零方法
	    fbEcCoESdoWriteHOffset: FB_EcCoESdoWrite                  ;           // 写COE 回零偏置
	    fbEcCoESdoWriteHVelo: FB_EcCoESdoWrite                    ;           // 写COE 回零速度
		
	     fbMcReadDistPerPulse: MC_ReadParameter;
	     fbMcReadGearRatio: MC_ReadParameter;
	     fbMcWritePosMonitorDisable: MC_WriteParameter;
	     fbMcWritePosMonitorEnable: MC_WriteParameter;
	         // 每脉冲移动量
	      lrDistPerPulse: LREAL := 0.0001;
	        // 减速比
	      lrGearRatio: LREAL := 1;
				udiHomeVelHigh: UDINT;
	      udiHomeVelLow: UDINT;
	      diHomeOffset: DINT;
		  bSDO:BOOL;
		  bSDOExe:BOOL;
		  Ton07: TON;
		  Ton61: TON;
		  Ton62: TON;
		  blink10ms:BLINK;
		  bPosMonitorDisabled: BOOL;
	      bPosMonitorAbled: BOOL;
END_VAR

posEdge_bCMD_HomeExecute(CLK:=bCMD_HomeExecute AND bCMD_EnableState AND NOT bResult_HomeError AND NOT bResult_HomeBusy);
ton_bCMD_HomeExecute(IN:=bCMD_HomeExecute,PT:=T#100MS);

IF posEdge_bCMD_HomeExecute.Q  THEN
	nStep:=1;
ELSIF	ton_bCMD_HomeExecute.Q THEN
	 bCMD_HomeExecute:=FALSE;
END_IF
// 超时定时器
ton_HomErr(IN:=bResult_HomeBusy , PT:=T#20S , Q=> , ET=> );
IF bCMD_siHomeMethod=0 AND bCMD_NegativeLimit AND ton_HomErr.Q THEN
		mcReset.Execute:=TRUE;
		nStep:=999;
ELSIF bCMD_siHomeMethod=1 AND bCMD_PositiveLimit AND ton_HomErr.Q THEN
		mcReset.Execute:=TRUE;
		nStep:=999;
END_IF
//触发读取写入SDO
			blink10ms(ENABLE:= , TIMELOW:= TIME#10MS , TIMEHIGH:= TIME#10MS , OUT=> bSDOExe);	
			IF nStep = 31 OR nStep = 35  THEN
				blink10ms.ENABLE := TRUE ; //循环触发，直到写入完成
			ELSE
				blink10ms.ENABLE := FALSE ;
			END_IF
			Ton07(IN:=( nStep = 15 OR nStep =20 OR  nStep = 25  OR nStep = 30), PT:=TIME#1000MS , Q=> , ET=> );
			Ton61(IN:=(nStep = 40),PT:=TIME#100MS,);
			Ton62(IN:=(nStep = 16),PT:=TIME#1000MS,);
			CASE nStep OF 
				1: 				    
					mcReset.Execute := FALSE ;
					nStep := 5 ;
				5: 
					bPosMonitorDisabled := TRUE;
					bPosMonitorAbled := FALSE;
					mcReset.Execute := TRUE ;
					IF mcReset.Done AND fbMcWritePosMonitorDisable.Done THEN
						mcReset.Execute := FALSE ;
						bPosMonitorDisabled := FALSE;
						nStep := 10 ;		 
					END_IF
				10:// 断使能
					 IF axis.Status.NotMoving AND axis.Status.StandStill THEN
                       bProcessPowerCtrl:=FALSE;
					   nStep := 15 ;
                     END_IF		 
				15:// 切换模式字，设定为6
					bCMD_siHomeMethod := 6 ;
					IF Ton07.Q  THEN
						nStep := 16 ;		 
					END_IF
				16: // 写入COE参数
				    bSDO:=TRUE;
					IF TON62.Q  THEN
						nStep:=20;
						bSDO:=FALSE;
					END_IF;
				20:// 重新使能
					 bProcessPowerCtrl:=TRUE;
					IF Ton07.Q AND bCMD_EnableState THEN
						nStep := 21;
					END_IF
				21:
					nStep := 25;
				25:// 复位
					mcReset.Execute := TRUE ;
					IF Ton07.Q AND mcReset.Done THEN
						nStep := 26;
					END_IF	
				26:// 	
						nStep:=30;
					
				30://					
					IF Ton07.Q THEN
						nStep := 31;
					END_IF;
				31:
					nStep :=35;
				35://等待状态字反馈 , 10 - Target Reached , 12 - Homing Attained , 13 - Homing Error
					IF uiStatusWord.10 AND uiStatusWord.12 AND NOT uiStatusWord.13 THEN
						mcReset.Execute :=TRUE;
						nStep:=36;
					END_IF
				36:
					IF mcReset.Done THEN
						mcReset.Execute := FALSE;
						bCMD_siHomeMethod :=8;
						nStep :=40;
					END_IF;
				40:	
					mcMoveAbs.Velocity:= REAL#2.0;
					IF Ton61.Q THEN
						mcMoveAbs.Execute:=TRUE;
					END_IF;
					IF mcMoveAbs.Done THEN
						mcMoveAbs.Execute:=FALSE;
						nStep := 50;	 
					END_IF	
				50:
					bPosMonitorDisabled := FALSE;
					bPosMonitorAbled := TRUE;
					IF fbMcWritePosMonitorEnable.Done THEN
						bPosMonitorAbled := FALSE;
						nStep := 60 ;
					END_IF;
				60:	
					bSDO:=FALSE;											
					bResult_HomeBusy := FALSE ;
					bResult_HomeDone := TRUE ;	
                    bResult_HomeError:= FALSE;				
					nStep := 0 ;		
				999:	 
				   	bSDO:=FALSE;											
					bResult_HomeBusy := FALSE ;
					bResult_HomeDone := FALSE ;
					bResult_HomeError:= TRUE;
					nStep := 0 ;	
			END_CASE	
ACT_AxisControl();
ACT_COE();
ACT_Reset();

ACTION ACT_AxisControl:
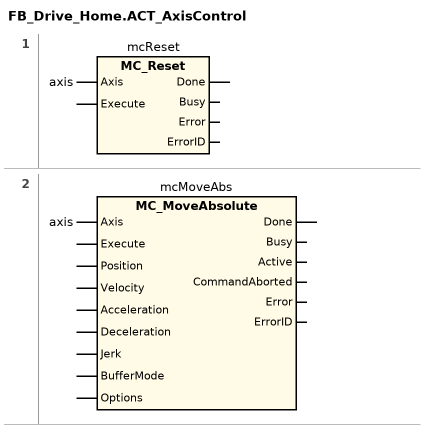
// NETWORK 1
mcReset(Axis := axis); // MC_Reset

// NETWORK 2
mcMoveAbs(Axis := axis); // MC_MoveAbsolute
END_ACTION

ACTION ACT_COE:

// 驱动器回零参数读取与写入	
	IF fbMcReadDistPerPulse.Valid AND fbMcReadGearRatio.Valid THEN
		udiHomeVelHigh := LREAL_TO_UDINT(rCMD_OffVelSetValue /(lrDistPerPulse / lrGearRatio));	
		udiHomeVelLow := LREAL_TO_UDINT(rCMD_TowardsVelSetValue /(lrDistPerPulse / lrGearRatio));
		diHomeOffset := LREAL_TO_DINT(rCMD_HomePosition /(lrDistPerPulse / lrGearRatio));
	END_IF;
		 
	//写入6098(HomingMethod)
	FB_EcCoESdoWrite_6098(
		sNetId:=stHomeCoEGroup.strNetID , 
		nSlaveAddr:=stHomeCoEGroup.wSlaveAddr , 
		nSubIndex:=16#00 , 
		nIndex:=16#6098 + (stHomeCoEGroup.uiAxisChannelNum - 1)*16#800  , 
		pSrcBuf:=ADR(bCMD_siHomeMethod) , 
		cbBufLen:=1 , 
		bExecute:= bSDO  , 
		tTimeout:= , 
		bBusy=> , 
		bError=> , 
		nErrId=> );

	//写入6099_01(HomeVelHigh)
	FB_EcCoESdoWrite_6099_01(
		sNetId:=stHomeCoEGroup.strNetID  , 
		nSlaveAddr:=stHomeCoEGroup.wSlaveAddr , 
		nSubIndex:=16#01 , 
		nIndex:=16#6099 + (stHomeCoEGroup.uiAxisChannelNum - 1)*16#800  , 
		pSrcBuf:=ADR(udiHomeVelHigh ) , 
		cbBufLen:=4 , 
		bExecute:= bSDO  , 
		tTimeout:= , 
		bBusy=> , 
		bError=> , 
		nErrId=> );	 
 
	//写入6099_02(HomeVelLow)
	FB_EcCoESdoWrite_6099_02(
		sNetId:=stHomeCoEGroup.strNetID   , 
		nSlaveAddr:=stHomeCoEGroup.wSlaveAddr , 
		nSubIndex:=16#02 , 
		nIndex:=16#6099 + (stHomeCoEGroup.uiAxisChannelNum- 1)*16#800  , 
		pSrcBuf:=ADR(udiHomeVelLow) , 
		cbBufLen:=4 , 
		bExecute:= bSDO , 
		tTimeout:= , 
		bBusy=> , 
		bError=> , 
		nErrId=> );

	//写入609A(HomeAcc)
//	FB_EcCoESdoWrite_609A(
//		sNetId:=stHomeCoEGroup.strNetID, 
//		nSlaveAddr:=stHomeCoEGroup.wSlaveAddr , 
//		nSubIndex:=16#00 , 
//		nIndex:=16#609A + (stHomeCoEGroup.uiAxisChannelNum - 1)*16#800  , 
//		pSrcBuf:=ADR(udiHomeAcc) , 
//		cbBufLen:=4 , 
//		bExecute:=bSDO , 
//		tTimeout:= , 
//		bBusy=> , 
//		bError=> , 
//		nErrId=> );	
	//写入607C (home offset）
	FB_EcCoESdoWrite_607C(
		sNetId:=stHomeCoEGroup.strNetID , 
		nSlaveAddr:=stHomeCoEGroup.wSlaveAddr , 
		nSubIndex:=16#00 , 
		nIndex:= 16#607C + (stHomeCoEGroup.uiAxisChannelNum - 1)*16#800 , 
		pSrcBuf:=ADR(diHomeOffset) , 
		cbBufLen:=SIZEOF(diHomeOffset) , 
		bExecute:=bSDO , 
		tTimeout:= , 
		bBusy=> , 
		bError=> , 
		nErrId=> );	
	//读取6041(Statusword)
	FB_EcCoESdoRead_6041(
		sNetId:=stHomeCoEGroup.strNetID , 
		nSlaveAddr:=stHomeCoEGroup.wSlaveAddr , 
		nSubIndex:=16#00 , 
		nIndex:=16#6041 + (stHomeCoEGroup.uiAxisChannelNum - 1)*16#800 , 
		pDstBuf:=ADR(uiStatusword) , 
		cbBufLen:=2 , 
		bExecute:=bSDOExe , 
		tTimeout:= , 
		bBusy=> , 
		bError=> , 
		nErrId=> );	
		
fbMcReadDistPerPulse(
	Axis:=axis , 
	Enable:= posEdge_bCMD_HomeExecute.Q, 
	ParameterNumber:=AxisEncoderScalingNumerator , 
	ReadMode:=READMODE_ONCE , 
	Value=>lrDistPerPulse );

fbMcReadGearRatio(
	Axis:= axis, 
	Enable:= posEdge_bCMD_HomeExecute.Q, 
	ParameterNumber:= AxisEncoderScalingDenominator,
	ReadMode:=READMODE_ONCE , 
	Value=>lrGearRatio );
	
fbMcWritePosMonitorEnable(
	Axis:=axis , 
	Execute:= bPosMonitorAbled, 
	ParameterNumber:= AxisEnPositionLagMonitoring, 
	Value:= 1, 
	Done=> , 
	Busy=> , 
	Error=> , 
	ErrorID=> );
fbMcWritePosMonitorDisable(
	Axis:= axis, 
	Execute:=bPosMonitorDisabled , 
	ParameterNumber:= AxisEnPositionLagMonitoring, 
	Value:= 0, 
	Done=> , 
	Busy=> , 
	Error=> , 
	ErrorID=> );
END_ACTION

ACTION ACT_Reset:
posEdge_bCMD_Reset(CLK:=bCMD_Reset);
ton_bCMD_Reset(IN:=bCMD_Reset,PT:=T#100MS);
ton_McReset(IN:=mcReset.Execute,PT:=T#100MS);
IF posEdge_bCMD_Reset.Q THEN
	bResult_HomeBusy:=FALSE;
	bResult_HomeDone:=FALSE;
	bResult_HomeError:=FALSE;
	nStep:=0;
	mcReset.Execute:=TRUE;
	mcMoveAbs.Execute:=FALSE;
ELSIF ton_bCMD_Reset.Q THEN
	bCMD_Reset:=FALSE;
END_IF

IF ton_McReset.Q THEN
	mcReset.Execute:=FALSE;
END_IF
END_ACTION

END_FUNCTION_BLOCK

// ---- FB/01_Axis/FB/FB_Axis_PE_Correct.TcPOU
FUNCTION_BLOCK FB_Axis_PE_Correct
VAR_IN_OUT
	AxisRef: AXIS_REF;
	// 补偿数据数组
	arstPitchTable: ARRAY[*] OF ST_CompensationElement;
END_VAR
VAR_INPUT
	// 功能开启
	bEnable: BOOL;
	// 轴回零状态
	bAxisHomeOK: BOOL;
	// 间隙补偿方向
	bBacklashDir: BOOL;
	// 间隙补偿
	rBcaklash: REAL;
	// 补偿间距
	rDistance: REAL;
END_VAR
VAR_OUTPUT
	// 当前补偿间隙值
	lrCurBacklash: LREAL;
	// 当前位置补偿值
	lrCOmpensation: LREAL;
	// 补偿功能运行状态
	bBusy: BOOL;
	// 错误
	bError: BOOL;
END_VAR
VAR
	strVersion: STRING;
	// TRUE
	bFirstRun: BOOL;
	i: DINT;
	mcBacklashCompensation: MC_BacklashCompensation;
	arstPitchTableConvert: ARRAY[0..999] OF ST_CompensationElement;
	stCompensationDesc: ST_CompensationDesc;
	fbPositionCompensation: FB_PositionCompensation;
	fbMcPositionCorrectionLimiter: MC_PositionCorrectionLimiter;
	fbMcReadParameter: MC_ReadParameter;
	fbMcWriteParaCompensationOff: MC_WriteParameter;
	fbMcWriteParaCompensationOn: MC_WriteParameter;
	bCompensationOn: BOOL;
	bCompensationOff: BOOL;
	tonCompensationOn: TON;
	tonCompensationOff: TON;
	i1: dINT;
	i2: dINT;
END_VAR
VAR_INPUT
	// 轴行程设置为0 到 负数，即点位越走越小时，置位True
	bAxisMovePosGetSmaller: BOOL;
END_VAR

(*********************
	by yu

	2023-12-29		设立运动轴位置补偿功能块
								位置补偿最大支持 1000 组补偿数据
								补偿位置从小到大,补偿值为误差值
	2025-07-11		增加版本记录
	2025-08-07		增加间隙补偿功能，背隙补偿开始的方向设定 bBacklashDir，根据轴的位置的移动方向确定，正向移动补偿为True，反向移动补偿为False
	2026-01-26		增加输入变量 bAxisMovePosGetSmaller ,当实际轴位置是越走越小时，此变量置为 true；轴位置是越走越大，置为 False
													
*********************)

strVersion := '2026-01-26';
IF bFirstRun THEN
	;
	bFirstRun := FALSE ;
END_IF


//根据输入补偿数据，对数据进行转换。数据抽取转换为定长数组
//超出输入数组大小的元素的补偿数据与最后一位数据的相同，补偿点位以等间距递增2
i1:= LOWER_BOUND(arstPitchTable,1);
i2:=UPPER_BOUND(arstPitchTable,1);
IF bAxisMovePosGetSmaller THEN //
	IF i2< 999 THEN
		FOR i:=(i2+1) TO 999 BY 1 DO
			arstPitchTableConvert[999-i].fPos := arstPitchTable[i2].fPos + rDistance *  DINT_TO_REAL((i - i2));
			arstPitchTableConvert[999-i].fCompensation := arstPitchTable[i2].fCompensation;
		END_FOR;
	END_IF;
	FOR i:=i1 TO i2 BY 1 DO
		arstPitchTableConvert[999-i].fPos := arstPitchTable[i].fPos;
		arstPitchTableConvert[999-i].fCompensation := arstPitchTable[i].fCompensation;
	END_FOR;
ELSE
	IF i2< 999 THEN
		FOR i:=(i2+1) TO 999 BY 1 DO
			arstPitchTableConvert[i].fPos := arstPitchTable[i2].fPos + rDistance *  DINT_TO_REAL((i - i2));
			arstPitchTableConvert[i].fCompensation := arstPitchTable[i2].fCompensation;
		END_FOR;
	END_IF;
	FOR i:=i1 TO i2 BY 1 DO
		arstPitchTableConvert[i].fPos := arstPitchTable[i].fPos;
		arstPitchTableConvert[i].fCompensation := arstPitchTable[i].fCompensation;
	END_FOR;	
END_IF

//补偿参数设定
stCompensationDesc.fPosMin:=arstPitchTableConvert[0].fPos;
stCompensationDesc.fPosMax:=arstPitchTableConvert[999].fPos;
stCompensationDesc.nTableElements:=1000;
stCompensationDesc.bModulo:=FALSE;

//轴参数中开启或关闭PositionCorrection功能
IF bEnable THEN
	bCompensationOff:=FALSE;
	tonCompensationOn(IN:= TRUE, PT:=TIME#10MS , Q=> , ET=> );
	IF tonCompensationOn.Q THEN
		bCompensationOn:=TRUE;
	END_IF	
ELSE
	bCompensationOn:=FALSE;		
	tonCompensationOff(IN:= TRUE, PT:=TIME#10MS , Q=> , ET=> );
	IF tonCompensationOff.Q THEN
		bCompensationOff:=TRUE;
	END_IF
END_IF



//功能块调用
//轴参数中开启PositionCorrection功能
fbMcWriteParaCompensationOn(
	Axis:= AxisRef, 
	Execute:= bCompensationOn, 
	ParameterNumber:=AxisEnablePosCorrection , 
	Value:= 1, 
	Done=> , 
	Busy=> , 
	Error=> , 
	ErrorID=> );
//轴参数中关闭PositionCorrection功能
fbMcWriteParaCompensationOff(
	Axis:= AxisRef, 
	Execute:= bCompensationOff, 
	ParameterNumber:=AxisEnablePosCorrection , 
	Value:=0 , 
	Done=> , 
	Busy=> , 
	Error=> , 
	ErrorID=> );
	

//间隙补偿功能必须在补偿功能开启后才可开启
IF fbMcReadParameter.Value = 1 THEN
	mcBacklashCompensation(
		Axis:= AxisRef, 
		Enable:= bAxisHomeOK AND bCompensationOn, 
		Backlash:= rBcaklash, 
		CompensationInPositiveDirection:= bBacklashDir, 
		Ramp:= , 
		DisableMode:= , 
		Options:= , 
		Enabled=> , 
		Busy=> , 
		Error=> , 
		ErrorID=> , 
		CurrentBacklash=> lrCurBacklash, 
		Limiting=> );
END_IF;
	
//获取位置补偿值功能块
fbPositionCompensation(
	Enable:=bAxisHomeOK AND bCompensationOn , 
	pTable:=ADR(arstPitchTableConvert) , 
	cbSize:=SIZEOF(arstPitchTableConvert) , 
	ReferenceAxis:= AxisRef.NcToPlc, 
	Desc:=stCompensationDesc , 
	Compensation=>lrCOmpensation , 
	Error=> , 
	ErrorId=> , 
	Active=> );

//在当前位置上写入补偿值功能块
fbMcPositionCorrectionLimiter(
	Axis:=AxisRef , 
	Enable:= bAxisHomeOK AND  bCompensationOn, 
	PositionCorrectionValue:= lrCOmpensation + lrCurBacklash, 
	CorrectionMode:=POSITIONCORRECTION_MODE_FAST  , 
	Acceleration:=500 , 
	CorrectionLength:= , 
	Busy=> , 
	Error=> , 
	ErrorID=> , 
	Limiting=> );	
	


//读取补偿功能开启状态
fbMcReadParameter(
	Axis:=AxisRef , 
	Enable:=TRUE , 
	ParameterNumber:= AxisEnablePosCorrection , 
	ReadMode:=READMODE_CYCLIC , 
	Valid=> , 
	Busy=> , 
	Error=> , 
	ErrorID=> , 
	Value=> );

//状态输出	
IF fbMcReadParameter.Valid THEN
	IF fbMcReadParameter.Value = 1 AND fbPositionCompensation.Active AND fbMcPositionCorrectionLimiter.Busy THEN
		bBusy:=TRUE;
	ELSE
		bBusy:=FALSE;
	END_IF;
END_IF;

END_FUNCTION_BLOCK

// ---- POUs/2_Nci/NCI_MAIN.TcPOU
PROGRAM NCI_MAIN
VAR 
 fbNci:FB_01_NCI;
 fbFalling :ARRAY[1..5] OF F_TRIG;
 fbRising  :ARRAY[1..5] OF R_TRIG;
 bEl5131_TrigH: BOOL;
 bEl5131_Trig : BOOL;
 bEl5131_TrigPressure: BOOL;
 tonWriteR:ARRAY [1..5] OF TON;
 bEl5131_ON :BOOL;
 stepWriteR:INT;
 
	tehn: INT;
END_VAR
VAR_IN_OUT
	
END_VAR

(*****************************************************************  
1.	out_stItpToPlc关联Channel2-inputs-FromPlc
    in_stItpToPlc 关联Channel2-output=ToPlc
2.  触发关联IO stIJP.bEx_TrigH/stIJP.bEx_Trig
*****************************************************************)
//底部真空破坏阀
IF Com_GVLS.bPlatformVacON THEN
	Y000002:=TRUE;
	Y000003:=FALSE;
END_IF

IF Com_GVLS.bPlatformVacOff THEN
	Y000002:=FALSE;
	Y000003:=TRUE;
END_IF

Y000001:=stIJP.bEx_TrigH OR bEl5131_TrigH  ;
Y000016:=(stIJP.bEx_Trig OR bEl5131_Trig )AND NOT stSystem.arErrorID[16];
stIJP.bEx_TrigHfb:=stIJP.bEx_TrigH OR bEl5131_TrigH ;

stIJP.bEx_Trigfb:=(stIJP.bEx_Trig OR bEl5131_Trig )AND NOT stSystem.arErrorID[16];
stIJP.bEx_TrigHfb:=stIJP.bEx_TrigH (*OR stIJP.bEl5131_Trig[1] OR stIJP_ZR.bEl5131_Trig *)(*AND  stSystem.arErrorID[15] AND   stSystem.arErrorID[16]
                      *)AND  stSystem.arErrorID[16];
stIJP.bEx_Trigfb:=(stIJP.bEx_Trig (*OR stIJP.bEl5131_Trig[1] OR stIJP_ZR.bEl5131_Trig *))(*AND  stSystem.arErrorID[15] AND   stSystem.arErrorID[16]
                      *)AND  stSystem.arErrorID[16];
					  
fbNci(
	stfbIJP:= stIJP, 
	in_stItpToPlc:= stIJP.in_stItpToPlc, 
	out_stItpToPlc:= stIJP.out_stItpToPlc, 
	nXAxisId:= arAXIS[1].NcToPlc.AxisId, 
	nYAxisId:= arAXIS[2].NcToPlc.AxisId, 
	nZAxisId:= arAXIS[4].NcToPlc.AxisId, 
	nQ1AxisId:= 0, 
	nQ2AxisId:= 0, 
	nChannelid:= stIJP.in_stItpToPlc.ChnId, 
	bProhibitMvALM:= );

IF stIJP.bStopExe THEN
   stIJP.bEx_TrigEl5131:=FALSE;
END_IF

// NCI报错监控 (error140-149)
stSystem.arErrorID[140+UDINT_TO_INT(stIJP.udiError)]:=stIJP.bError;

ACTION ACTNCIDispenser:
stIJP.strPRGName:=' 点胶XYZ插补';
stIJP.lrOverrideSet:=100;
(* IO关联*)
// NC:=stIJP.bEx_Trig;
stIJP.iJetOnDelay:=1;
END_ACTION

END_PROGRAM

// ---- FB/02_NCI/FB/FB_01_NCI.TcPOU

FUNCTION_BLOCK FB_01_NCI
// 定义功能块FB_01_NCI，用于数控指令(NCI)的集中控制

VAR_IN_OUT
  stfbIJP         :ST_IJP;  // 输入输出变量，ST_IJP结构体，用于与外部交换数据
  in_stItpToPlc :   NCTOPLC_NCICHANNEL_REF;
  out_stItpToPlc :  PLCTONC_NCICHANNEL_REF;
END_VAR

VAR_INPUT
	nXAxisId:UDINT;
	nYAxisId:UDINT;
	nZAxisId:UDINT;
	nQ1AxisId:UDINT;
	nQ2AxisId:UDINT;
	nChannelid:UDINT;
	bProhibitMvALM:BOOL;
END_VAR

VAR
  // 声明内部使用的功能块变量
  fbBuildGroup  :FB_02_BuidGroup;    // 用于构建运动组的功能块
  fbLoadProg    :FB_03_LoadProg;     // 用于加载程序的功能块
  fbStart       :FB_04_Start;        // 用于启动运动的功能块
  fbExStop      :FB_06_ExSTOP;       // 用于紧急停止的功能块
  fbAfterStop   :FB_012_StepOnAfterStopEx;  // 用于紧急停止后处理的功能块
  fbReset       :FB_08_ReSetEx;      // 用于复位系统的功能块
  fbSetoverride :FB_09_SetOverridePercent;  // 用于设置速度百分比的功能块
  fbClearGrp    :FB_05_ClearGrp;     // 用于清除运动组的功能块
  fbFastMFunc   :FB_07_FastMFunc;    // 用于快速M功能的功能块
  WriteRParameter:FB_011WriteRParameter;  // 用于写入R参数的功能块
  ReadRParameter:FB_010_ReadRParameter;   // 用于读取R参数的功能块
  fbItpEStopEx: ItpEStopEx ;    // 暂停G代码运行
  fbItpStepOnAfterEStopEx : ItpStepOnAfterEStopEx ;  // 暂停G代码后继续执行G代码
  arrfbSetAlarm:ARRAY [1..6] OF FB_SetError;
	// 报错
	a: BOOL;  //  程序加载错误
	b: BOOL; //  启动错误
	c: BOOL; // 停止错误
	d: BOOL; // 停止后在继续错误
	e: BOOL; // 复位出错
	f: BOOL;  // 创建运动轴错误
	g: BOOL;  // 清除运动轴错误
 posEdge_bCMD_bWriteRParExe:R_TRIG;
 ton_bCMD_bWriteRParExe:TON;
 ton_bCMD_bReadRParExe:blink;
 posEdge_bCMD_bLoadPgmExe:R_TRIG;
 ton_bCMD_bLoadPgmExe:TON;
 posEdge_bCMD_bBuildGroupExe:R_TRIG;
 ton_bCMD_bBuildGroupExe:TON;
 posEdge_bCMD_bClearGroupExe:R_TRIG;
 ton_bCMD_bClearGroupExe:TON;
 fbWriteZeroShift: FB_013_WriteZeroShiftEx;
END_VAR


// 调用快速M功能功能块
// 参数说明：
// stfbIJP07: 传递ST_IJP结构体数据
// stItpToPlc: 从ITP(Interpreter)到PLC的数据流
// stPlcToItp: 从PLC到ITP的数据流

fbFastMFunc(stfbIJP07:=stfbIJP, stItpToPlc:= in_stItpToPlc, stPlcToItp:= out_stItpToPlc);	

// 调用写入R参数功能块
// 参数说明：
// Execute: 执行信号，来自stfbIJP.bWriteRParExe
// nRParamAry: 要写入的R参数数组，来自stfbIJP.arrWriteRPar
posEdge_bCMD_bWriteRParExe(CLK:=stfbIJP.bWriteRParExe);
ton_bCMD_bWriteRParExe(IN:=stfbIJP.bWriteRParExe,PT:=T#100MS);
WriteRParameter(Execute:= stfbIJP.bWriteRParExe,fbnChannelid:=nChannelid, nRParamAry:= stfbIJP.arrWriteRPar);

// 调用读取R参数功能块
// 参数说明：
// Execute: 执行信号，来自stfbIJP.bReadRParExe
// nRParamAry: 读取的R参数数组，输出到stfbIJP.arrReadRPar
ton_bCMD_bReadRParExe(ENABLE:=stfbIJP.bReadRParExe,TIMEHIGH:=T#50MS,TIMELOW:=T#50MS,OUT=>);
ReadRParameter(Execute:= ton_bCMD_bReadRParExe.OUT,fbnChannelid:=nChannelid, nRParamAry=> stfbIJP.arrReadRPar);

(******************* NCI功能块调用部分 **************)
// 调用速度百分比设置功能块
// 参数说明：
// OverridePercent: 速度百分比值，来自stfbIJP.lrOverrideSet

fbSetoverride(
    OverridePercent:= stfbIJP.lrOverrideSet,
    stItpToPlc:= in_stItpToPlc,
    stPlcToItp:= out_stItpToPlc );

// 调用构建运动组功能块
// 参数说明：
// bExecute: 构建组执行信号，来自stfbIJP.bBuildGroupExe
posEdge_bCMD_bBuildGroupExe(CLK:=stfbIJP.bBuildGroupExe);
ton_bCMD_bBuildGroupExe(IN:=stfbIJP.bBuildGroupExe,PT:=T#100MS);
IF ton_bCMD_bBuildGroupExe.Q THEN
	stfbIJP.bBuildGroupExe:=FALSE;
END_IF
fbBuildGroup(
    bExecute:= stfbIJP.bBuildGroupExe, 
    bBusy=> , 
    bError=> f, 
    bDone=> , 
    nXAxisId:= nXAxisId, 
    nYAxisId:= nYAxisId, 
    nZAxisId:= nZAxisId, 
	nQ1AxisId:= nQ1AxisId, 
	nQ2AxisId:= nQ2AxisId, 
    stItpToPlc:=  in_stItpToPlc, 
    stPlcToItp:= out_stItpToPlc);

// 调用清除运动组功能块
// 参数说明：
// bExecute: 清除组执行信号，来自stfbIJP.bClearGroupExe
posEdge_bCMD_bClearGroupExe(CLK:=stfbIJP.bClearGroupExe);
ton_bCMD_bClearGroupExe(IN:=stfbIJP.bClearGroupExe,PT:=T#100MS);
IF ton_bCMD_bClearGroupExe.Q THEN
	stfbIJP.bClearGroupExe:=FALSE;
END_IF
fbClearGrp(
    bExecute:= stfbIJP.bClearGroupExe, 
    bBusy=> , 
    bError=> g, 
    bDone=> , 
    stItpToPlc:= in_stItpToPlc, 
    stPlcToItp:= out_stItpToPlc);
// 调用加载程序功能块
// 参数说明：
// bExecute: 执行信号，来自stfbIJP.bLoadPGMExe
// sPrgName: 程序名称，来自stfbIJP.strPRGName
// bError: 错误状态，输出到stfbIJP.bError
// bDone: 完成状态，输出到stfbIJP.bLoadPGMDone
// stX/Y/Z: 传递各轴控制接口
// stItpToPlc/stPlcToItp: 数据流接口
posEdge_bCMD_bLoadPgmExe(CLK:=stfbIJP.bLoadPGMExe);
ton_bCMD_bLoadPgmExe(IN:=stfbIJP.bLoadPGMExe,PT:=T#100MS);
IF ton_bCMD_bLoadPgmExe.Q THEN
	stfbIJP.bLoadPGMExe:=FALSE;
END_IF
fbLoadProg(
    bExecute:= stfbIJP.bLoadPGMExe, 
    sPrgName:= stfbIJP.strPRGName, 
    bBusy=> , 
    bError=> a, 
    bDone=> stfbIJP.bLoadPGMDone, 
    stItpToPlc:= in_stItpToPlc, 
    stPlcToItp:= out_stItpToPlc);

// 调用启动功能块
// 参数说明：
// bExecute: 启动执行信号，来自stfbIJP.bStartExe
// bExecute1: 停止执行信号，来自stfbIJP.bStopExe
// bError: 错误状态，输出到stfbIJP.bError

fbStart(
    bExecute:= stfbIJP.bStartExe , 
    bExecute1:= stfbIJP.bStopExe, 
    bBusy=> ,
    bError=> b, 
    bDone=> ,  
    stItpToPlc:= in_stItpToPlc, 
    stPlcToItp:= out_stItpToPlc);

// 调用紧急停止功能块
// 参数说明：
// bExecute: 紧急停止执行信号，来自stfbIJP.bEstopExe

fbExStop(
    bExecute:= stfbIJP.bEstopExe, 
    bBusy=> , 
    bError=> c, 
    bDone=> , 
    stItpToPlc:=  in_stItpToPlc, 
    stPlcToItp:=  out_stItpToPlc);
IF fbExStop.bDone THEN
	stfbIJP.bEstopExe:=FALSE;
	stfbIJP.bEx_TrigH:=FALSE;	
	stfbIJP.bEx_Trig:=FALSE;	
END_IF
// 调用紧急停止后处理功能块
// 参数说明：
// bExecute: 执行信号，来自stfbIJP.bAfterEstopExe

fbAfterStop(
    bExecute:= stfbIJP.bAfterEstopExe, 
    bBusy=> , 
    bError=> d, 
    bDone=> , 
    stItpToPlc:= in_stItpToPlc, 
    stPlcToItp:= out_stItpToPlc);
IF fbAfterStop.bDone THEN
	stfbIJP.bAfterEstopExe:=FALSE;
END_IF
// 调用复位功能块
// 参数说明：
// bExecute: 复位执行信号，来自stfbIJP.bResetExe

fbReset(
    bExecute:= stfbIJP.bResetExe, 
    bBusy=> , 
    bError=> e, 
    bDone=> , 
    stItpToPlc:= in_stItpToPlc, 
    stPlcToItp:= out_stItpToPlc);
IF fbReset.bDone THEN
	stfbIJP.bResetExe:=FALSE;
END_IF
	
	// 暂停G代码运行
fbItpEStopEx(
	sNciToPlc:= in_stItpToPlc, 
	bExecute:= stfbIJP.bItpEStopEx , 
	fDec:= , 
	fJerk:= , 
	tTimeOut:= T#300MS, 
	bBusy=> , 
	bErr=> stfbIJP.bErrorEStop, 
	nErrId=> );
	// 暂停G代码后继续执行G代码
fbItpStepOnAfterEStopEx(
	bExecute:= stfbIJP.bItpStepOnAfterEStopEx , 
	tTimeOut:= T#300MS, 
	sNciToPlc:= in_stItpToPlc, 
	bBusy=> , 
	bErr=> stfbIJP.bErrorEStop,   
	nErrId=> );
	
fbWriteZeroShift(
	bExecute:=stfbIJP.bWriteZeroShiftExe , 
	nZsNo:=54 , 
	tTimeOut:=T#300MS , 
	lZeroShiftX:=stfbIJP.lZeroShiftX , 
	lZeroShiftY:=stfbIJP.lZeroShiftY , 
	lZeroShiftZ:=stfbIJP.lZeroShiftZ , 
	bBusy=> , 
	bErr=> , 
	nErrId=> , 
	stItpToPlc:=in_stItpToPlc );	
	
	IF a OR b OR c OR d OR e OR f OR g THEN 
		stfbIJP.bError:= TRUE;
		ELSE 
			stfbIJP.bError:= FALSE;
		END_IF

	
// 错误状态处理逻辑
// 根据各功能块的错误状态设置全局错误代码
IF  fbLoadProg.bError THEN
    stfbIJP.udiError:=1;  // 加载程序错误
ELSIF fbStart.bError THEN
    stfbIJP.udiError:=2;  // 启动错误
ELSIF fbExStop.bError THEN
    stfbIJP.udiError:=3;  // 紧急停止错误
ELSIF fbReset.bError THEN
    stfbIJP.udiError:=4;  // 复位错误
ELSIF fbBuildGroup.bError THEN
    stfbIJP.udiError:=5;  // 构建组错误
ELSIF fbClearGrp.bError THEN
    stfbIJP.udiError:=6;  // 清除组错误	
ELSE
    stfbIJP.udiError:=0;  // 无错误	
END_IF
// 加载程序错误
arrfbSetAlarm[1](
	bEnable:= TRUE, 
	iErrorID:= 130+6*(UINT_TO_INT(in_stItpToPlc.ChnId)-2), 
	bExecute:= stfbIJP.arErrorID[1], 
	bReset:= stSystem.bReset, 
	strErrorInfoEN:= 'Load Err', 
	wstrErrorInfoCN:="加载程序错误" , 
	enumErrorClass:= 6, 
	wstr1:=STRING_TO_WSTRING(stfbIJP.strNciName),
	D1:=UDINT_TO_DINT(in_stItpToPlc.ErrorCode),
    );
// 启动错误
arrfbSetAlarm[2](
	bEnable:= TRUE, 
	iErrorID:= 130+6*(UINT_TO_INT(in_stItpToPlc.ChnId)-2)+1, 
	bExecute:= stfbIJP.arErrorID[1], 
	bReset:= stSystem.bReset, 
	strErrorInfoEN:= 'Start Err', 
	wstrErrorInfoCN:="加载程序错误" , 
	enumErrorClass:= 6, 
	wstr1:=STRING_TO_WSTRING(stfbIJP.strNciName),
	D1:=UDINT_TO_DINT(in_stItpToPlc.ErrorCode),
    );
// 紧急停止错误
arrfbSetAlarm[3](
	bEnable:= TRUE, 
	iErrorID:= 130+6*(UINT_TO_INT(in_stItpToPlc.ChnId)-2)+2, 
	bExecute:= stfbIJP.arErrorID[1], 
	bReset:= stSystem.bReset, 
	strErrorInfoEN:= 'Estop Err', 
	wstrErrorInfoCN:="紧急停止错误" , 
	enumErrorClass:= 6, 
	wstr1:=STRING_TO_WSTRING(stfbIJP.strNciName),
	D1:=UDINT_TO_DINT(in_stItpToPlc.ErrorCode),
    );
// 复位错误
arrfbSetAlarm[4](
	bEnable:= TRUE, 
	iErrorID:= 130+6*(UINT_TO_INT(in_stItpToPlc.ChnId)-2)+3, 
	bExecute:= stfbIJP.arErrorID[1], 
	bReset:= stSystem.bReset, 
	strErrorInfoEN:= 'Reset Err', 
	wstrErrorInfoCN:="复位错误" , 
	enumErrorClass:= 6, 
	wstr1:=STRING_TO_WSTRING(stfbIJP.strNciName),
	D1:=UDINT_TO_DINT(in_stItpToPlc.ErrorCode),
    );
// 构建组错误
arrfbSetAlarm[5](
	bEnable:= TRUE, 
	iErrorID:= 130+6*(UINT_TO_INT(in_stItpToPlc.ChnId)-2)+4, 
	bExecute:= stfbIJP.arErrorID[1], 
	bReset:= stSystem.bReset, 
	strErrorInfoEN:= 'Build Err', 
	wstrErrorInfoCN:="构建组错误" , 
	enumErrorClass:= 6, 
	wstr1:=STRING_TO_WSTRING(stfbIJP.strNciName),
	D1:=UDINT_TO_DINT(in_stItpToPlc.ErrorCode),
    );
// 清除组错误
arrfbSetAlarm[6](
	bEnable:= TRUE, 
	iErrorID:= 130+6*(UINT_TO_INT(in_stItpToPlc.ChnId)-2)+4, 
	bExecute:= stfbIJP.arErrorID[1], 
	bReset:= stSystem.bReset, 
	strErrorInfoEN:= 'Clear Err', 
	wstrErrorInfoCN:="清除组错误" , 
	enumErrorClass:= 6, 
	wstr1:=STRING_TO_WSTRING(stfbIJP.strNciName),
	D1:=UDINT_TO_DINT(in_stItpToPlc.ErrorCode),
    );

END_FUNCTION_BLOCK

// ---- FB/02_NCI/FB/FB_02_BuidGroup.TcPOU
FUNCTION_BLOCK FB_02_BuidGroup

VAR_INPUT
	bExecute:BOOL;
	nXAxisId:UDINT;
	nYAxisId:UDINT;
	nZAxisId:UDINT;
	nQ1AxisId:UDINT;
	nQ2AxisId:UDINT;
END_VAR
VAR_OUTPUT
	bBusy:BOOL;(*功能块执行忙标志*)
	bError:BOOL;(*出错*)
	bDone:BOOL;(*执行完毕*)
END_VAR
VAR_IN_OUT
//	stX:AXIS_REF;
//	stY:AXIS_REF;
//	stZ:AXIS_REF;
	stItpToPlc :NCTOPLC_NCICHANNEL_REF;
	stPlcToItp:PLCTONC_NCICHANNEL_REF;
END_VAR
VAR
	BuidGroupStep:INT:=0;
	fbBuidGroup:CfgBuildExt3DGroup;(*配置NciGroup*)
END_VAR

CASE BuidGroupStep OF
	0:
	  IF  bExecute THEN
		 bBusy:=TRUE;(*FB执行状态*)
		  bDone:=FALSE;(*FB执行完毕*)
		  bError:=FALSE;(*报错*)
		  BuidGroupStep:=10;(*进入10步*) 
	  END_IF
	10:
	  fbBuidGroup(
	    bExecute:= TRUE, 
	    nGroupId:= ItpGetGroupId(sNciToPlc:=stItpToPlc), 
	    nXAxisId:= nXAxisId, 
	    nYAxisId:= nYAxisId, 
	    nZAxisId:= nZAxisId, 
	    nQ1AxisId:= nQ1AxisId, 
	    nQ2AxisId:= nQ2AxisId, 
	    nQ3AxisId:= 0, 
	    nQ4AxisId:= 0, 
	    nQ5AxisId:= 0, 
	    tTimeOut:= , 
	    bBusy=> , 
	    bErr=> , 
	    nErrId=> );
	   IF NOT fbBuidGroup.bBusy THEN
		  IF NOT fbBuidGroup.bErr THEN
			BuidGroupStep:=20;(*进入20步*)  
		  ELSE
			bBusy:=FALSE;
			bError:=TRUE;
			BuidGroupStep:=999;
		  END_IF
		fbBuidGroup(bExecute:= FALSE,nGroupId:= ItpGetGroupId(sNciToPlc:=stItpToPlc));
	    END_IF
	 20:
	   //ItpSetOverridePercent(fOverridePercent:= 100, sPlcToNci:= stPlcToItp);
	   bDone:=TRUE;
       bBusy:=FALSE;   
	   IF NOT bExecute THEN
		 BuidGroupStep:=0;
	   END_IF
	 999:
	   IF NOT bExecute THEN		   
	    BuidGroupStep:=0;
        bError:=FALSE; 
	 END_IF
END_CASE

END_FUNCTION_BLOCK

// ---- FB/02_NCI/FB/FB_03_LoadProg.TcPOU
FUNCTION_BLOCK FB_03_LoadProg
VAR_INPUT
	bExecute:BOOL;
	sPrgName:STRING(255);(*G代码链接*)
//	nXAxisId:UDINT;
//	nYAxisId:UDINT;
//	nZAxisId:UDINT;
END_VAR
VAR_OUTPUT
	bBusy:BOOL;(*功能块执行忙标志*)
	bError:BOOL;(*出错*)
	bDone:BOOL;(*执行完毕*)
END_VAR
VAR_IN_OUT
//	stX:AXIS_REF;
//	stY:AXIS_REF;
//	stZ:AXIS_REF;
	stItpToPlc :NCTOPLC_NCICHANNEL_REF;
	stPlcToItp:PLCTONC_NCICHANNEL_REF;
END_VAR
VAR
	LoadProgStep:INT:=0;
	fbLoadProg:ItpLoadProgEx;(*下载NCI程序*)
END_VAR

sPrgName := Com_GVLS.stIJP.strNciName;

CASE LoadProgStep OF
	0:
	  IF  bExecute THEN
//		  LoadProgDone:=FALSE;
		  bBusy:=TRUE;(*FB执行状态*)
		  bDone:=FALSE;(*FB执行完毕*)
		  bError:=FALSE;(*报错*)
		  LoadProgStep:=10;(*进入10步*) 
	  END_IF
	10:
	   fbLoadProg(
	    sNciToPlc:= stItpToPlc, 
	    bExecute:= TRUE, 
	    sPrg:= sPrgName, 
	    nLength:= INT_TO_UDINT(LEN(sPrgName)), 
	    tTimeOut:= , 
	    bBusy=> , 
	    bErr=> , 
	    nErrId=> );
	   IF NOT fbLoadProg.bBusy THEN
		  IF NOT fbLoadProg.bErr THEN
			LoadProgStep:=20;(*进入20步*)  
		  ELSE
			bBusy:=FALSE;
			bError:=TRUE;
			LoadProgStep:=999;
		  END_IF
		 fbLoadProg(sNciToPlc:= stItpToPlc,bExecute:= FALSE,sPrg:= sPrgName,nLength:= INT_TO_UDINT(LEN(sPrgName)));
		//fbLoadProg.bExecute:=FALSE;  
//fbLoadProg(
	   //  sNciToPlc:= stItpToPlc, 
	   //  bExecute:= FALSE);
	    END_IF
	 20:
	   bDone:=TRUE;
       bBusy:=FALSE;  
//       LoadProgDone:=TRUE; 
	   IF NOT bExecute THEN
	//	 fbLoadProg.bExecute:=FALSE;   
		 LoadProgStep:=0;
	   END_IF
	 999:
	   IF NOT bExecute THEN		   
	    LoadProgStep:=0;
        bError:=FALSE; 
	   END_IF
END_CASE

END_FUNCTION_BLOCK

// ---- FB/02_NCI/FB/FB_04_Start.TcPOU
FUNCTION_BLOCK FB_04_Start
VAR_INPUT
	bExecute:BOOL;
	bExecute1:BOOL;
END_VAR
VAR_OUTPUT
	bBusy:BOOL;(*功能块执行忙标志*)
	bError:BOOL;(*出错*)
	bDone:BOOL;(*执行完毕*)
END_VAR
VAR_IN_OUT
//	stX:AXIS_REF;
//	stY:AXIS_REF;
//	stZ:AXIS_REF;
	stItpToPlc :NCTOPLC_NCICHANNEL_REF;
	stPlcToItp:PLCTONC_NCICHANNEL_REF;
END_VAR
VAR
	StartStep:INT:=0;
	fbStart:ItpStartStopEx;(*启动和停止*)
END_VAR

CASE StartStep OF
	0:
	  IF  bExecute OR bExecute1 THEN
		 bBusy:=TRUE;(*FB执行状态*)
		 bDone:=FALSE;(*FB执行完毕*)
		 bError:=FALSE;(*报错*)
		 StartStep:=10;(*进入10步*) 
	  END_IF
	10:
	  fbStart(
     	bStart:= bExecute, 
	    bStop:= bExecute1, 
	    tTimeOut:= , 
	    sNciToPlc:= stItpToPlc, 
	    bBusy=> , 
	    bErr=> , 
	    nErrId=> );
	   IF NOT fbStart.bBusy THEN
		  IF NOT fbStart.bErr THEN
			StartStep:=20;(*进入20步*)  
		  ELSE
			bBusy:=FALSE;
			bError:=TRUE;
			StartStep:=999;
		  END_IF
		  fbStart(bStart:= FALSE,bStop:=FALSE,sNciToPlc:= stItpToPlc); 
	    END_IF
	 20:
	   bDone:=TRUE;
       bBusy:=FALSE;   
	   IF NOT bExecute AND NOT bExecute1 THEN
		 StartStep:=0;
	   END_IF
	 999:
	   IF NOT bExecute AND NOT bExecute1 THEN		   
	    StartStep:=0;
        bError:=FALSE; 
	   END_IF
END_CASE

END_FUNCTION_BLOCK

// ---- FB/02_NCI/FB/FB_06_ExSTOP.TcPOU
FUNCTION_BLOCK FB_06_ExSTOP
VAR_INPUT
	bExecute:BOOL;
END_VAR
VAR_OUTPUT
	bBusy:BOOL;(*功能块执行忙标志*)
	bError:BOOL;(*出错*)
	bDone:BOOL;(*执行完毕*)
END_VAR
VAR_IN_OUT
//	stX:AXIS_REF;
//	stY:AXIS_REF;
//	stZ:AXIS_REF;
	stItpToPlc :NCTOPLC_NCICHANNEL_REF;
	stPlcToItp:PLCTONC_NCICHANNEL_REF;
END_VAR
VAR
	StopStep:INT:=0;
	fbEStop:ItpEStopEx;(*暂停*)
END_VAR

CASE StopStep OF
	0:
	  IF  bExecute THEN
		 bBusy:=TRUE;(*FB执行状态*)
		 bDone:=FALSE;(*FB执行完毕*)
		 bError:=FALSE;(*报错*)
		 StopStep:=10;(*进入10步*) 
	  END_IF
	10:
	  fbEStop(
	    sNciToPlc:=stItpToPlc , 
	    bExecute:= TRUE, 
	    fDec:= 40000, 
	    fJerk:= 40000, 
	    tTimeOut:= , 
	    bBusy=> , 
	    bErr=> , 
	    nErrId=> );
	   IF NOT fbEStop.bBusy THEN
		  IF NOT fbEStop.bErr THEN
			StopStep:=20;(*进入20步*)  
		  ELSE
			bBusy:=FALSE;
			bError:=TRUE;
			StopStep:=999;
		  END_IF
		  fbEStop(bExecute:= FALSE,sNciToPlc:= stItpToPlc); 
	    END_IF
	 20:
	   bDone:=TRUE;
       bBusy:=FALSE;   
	   IF NOT bExecute THEN
		 StopStep:=0;
	   END_IF
	 999:
	   IF NOT bExecute THEN		   
	    StopStep:=0;
        bError:=FALSE; 
	   END_IF
END_CASE

END_FUNCTION_BLOCK

// ---- FB/02_NCI/FB/FB_012_StepOnAfterStopEx.TcPOU
FUNCTION_BLOCK FB_012_StepOnAfterStopEx

VAR_INPUT
	bExecute:BOOL;
END_VAR
VAR_OUTPUT
	bBusy:BOOL;(*功能块执行忙标志*)
	bError:BOOL;(*出错*)
	bDone:BOOL;(*执行完毕*)
END_VAR
VAR_IN_OUT
//	stX:AXIS_REF;
//	stY:AXIS_REF;
//	stZ:AXIS_REF;
	stItpToPlc :NCTOPLC_NCICHANNEL_REF;
	stPlcToItp:PLCTONC_NCICHANNEL_REF;
END_VAR
VAR
	AfterStopStep:INT:=0;
	fbsteponafterestop:ItpStepOnAfterEStopEx;(*暂停重启*)
END_VAR

CASE AfterStopStep OF
	0:
	  IF  bExecute THEN
		 bBusy:=TRUE;(*FB执行状态*)
		 bDone:=FALSE;(*FB执行完毕*)
		 bError:=FALSE;(*报错*)
		 AfterStopStep:=10;(*进入10步*) 
	  END_IF
	10:
	  fbsteponafterestop(
	    bExecute:= TRUE, 
	    tTimeOut:= , 
	    sNciToPlc:= stItpToPlc, 
	    bBusy=> , 
	    bErr=> , 
	    nErrId=> );
	   IF NOT fbsteponafterestop.bBusy THEN
		  IF NOT fbsteponafterestop.bErr THEN
			AfterStopStep:=20;(*进入20步*)  
		  ELSE
			bBusy:=FALSE;
			bError:=TRUE;
			AfterStopStep:=999;
		  END_IF
		  fbsteponafterestop(bExecute:= FALSE,sNciToPlc:= stItpToPlc); 
	    END_IF
	 20:
	   bDone:=TRUE;
       bBusy:=FALSE;   
	   IF NOT bExecute THEN
		 AfterStopStep:=0;
	   END_IF
	 999:
	   IF NOT bExecute THEN		   
	    AfterStopStep:=0;
        bError:=FALSE; 
	   END_IF
END_CASE

END_FUNCTION_BLOCK

// ---- FB/02_NCI/FB/FB_08_ReSetEx.TcPOU
FUNCTION_BLOCK FB_08_ReSetEx
VAR_INPUT
	bExecute:BOOL;
END_VAR
VAR_OUTPUT
	bBusy:BOOL;(*功能块执行忙标志*)
	bError:BOOL;(*出错*)
	bDone:BOOL;(*执行完毕*)
END_VAR
VAR_IN_OUT
//	stX:AXIS_REF;
//	stY:AXIS_REF;
//	stZ:AXIS_REF;
	stItpToPlc :NCTOPLC_NCICHANNEL_REF;
	stPlcToItp:PLCTONC_NCICHANNEL_REF;
END_VAR
VAR
	ResetStep:INT:=0;
	fbReset:ItpResetEx2;(*启动和停止*)
END_VAR

CASE ResetStep OF
	0:
	  IF  bExecute THEN
		 bBusy:=TRUE;(*FB执行状态*)
		 bDone:=FALSE;(*FB执行完毕*)
		 bError:=FALSE;(*报错*)
		 ResetStep:=10;(*进入10步*) 
	  END_IF
	10:
	  fbReset(
	    bExecute:= TRUE, 
	    tTimeOut:=, 
	    sNciToPlc:= stItpToPlc, 
	    bBusy=> , 
	    bErr=> , 
	    nErrId=> );
	   IF NOT fbReset.bBusy THEN
		  IF NOT fbReset.bErr THEN
			ResetStep:=20;(*进入20步*)  
		  ELSE
			bBusy:=FALSE;
			bError:=TRUE;
			ResetStep:=999;
		  END_IF
		  fbReset(bExecute:= FALSE,sNciToPlc:= stItpToPlc); 
	    END_IF
	 20:
	   bDone:=TRUE;
       bBusy:=FALSE;   
	   IF NOT bExecute THEN
		 ResetStep:=0;
	   END_IF
	 999:
	   IF NOT bExecute THEN		   
	    ResetStep:=0;
        bError:=FALSE; 
	   END_IF
END_CASE

END_FUNCTION_BLOCK

// ---- FB/02_NCI/FB/FB_09_SetOverridePercent.TcPOU
FUNCTION_BLOCK FB_09_SetOverridePercent
VAR_INPUT
	OverridePercent:LREAL:=100;
END_VAR
VAR_OUTPUT
END_VAR
VAR_IN_OUT
	stItpToPlc :NCTOPLC_NCICHANNEL_REF;
	stPlcToItp:PLCTONC_NCICHANNEL_REF;
END_VAR
VAR
END_VAR

ItpSetOverridePercent(fOverridePercent:= OverridePercent, sPlcToNci:= stPlcToItp);

END_FUNCTION_BLOCK

// ---- FB/02_NCI/FB/FB_05_ClearGrp.TcPOU
FUNCTION_BLOCK FB_05_ClearGrp
VAR_INPUT
	bExecute:BOOL;
END_VAR
VAR_OUTPUT
	bBusy:BOOL;(*功能块执行忙标志*)
	bError:BOOL;(*出错*)
	bDone:BOOL;(*执行完毕*)
END_VAR
VAR_IN_OUT
//	stX:AXIS_REF;
//	stY:AXIS_REF;
//	stZ:AXIS_REF;
	stItpToPlc :NCTOPLC_NCICHANNEL_REF;
	stPlcToItp:PLCTONC_NCICHANNEL_REF;
END_VAR
VAR
	ClearGrp:INT:=0;
	fbClearGrp:CfgReconfigGroup;(*清除NciGroup*)
END_VAR

CASE ClearGrp OF
	0:
	  IF  bExecute THEN
		 bBusy:=TRUE;(*FB执行状态*)
		 bDone:=FALSE;(*FB执行完毕*)
		 bError:=FALSE;(*报错*)
		 ClearGrp:=10;(*进入10步*) 
	  END_IF
	10:
	  fbClearGrp(
 	    bExecute:= TRUE, 
	    nGroupId:= ItpGetGroupId(sNciToPlc:=stItpToPlc), 
	    tTimeOut:= , 
	    bBusy=> , 
	    bErr=> , 
	    nErrId=> );
	   IF NOT fbClearGrp.bBusy THEN
		  IF NOT fbClearGrp.bErr THEN
			ClearGrp:=20;(*进入20步*)  
		  ELSE
			bBusy:=FALSE;
			bError:=TRUE;
			ClearGrp:=999;
		  END_IF
		fbClearGrp(bExecute:= FALSE,nGroupId:= ItpGetGroupId(sNciToPlc:=stItpToPlc));
	    END_IF
	 20:
	   bDone:=TRUE;
       bBusy:=FALSE; 
	   IF NOT bExecute THEN
		 ClearGrp:=0;
	   END_IF
	 999:
	   IF NOT bExecute THEN		   
	    ClearGrp:=0;
        bError:=FALSE; 
	   END_IF
END_CASE

END_FUNCTION_BLOCK

// ---- FB/02_NCI/FB/FB_07_FastMFunc.TcPOU
FUNCTION_BLOCK FB_07_FastMFunc
//VAR_INPUT
//	EX_Trigtime:INT;
//	bLayerChanged:BOOL; // 切换指令
//END_VAR   
//VAR_OUTPUT
//	EX_TrigH:BOOL;       // 
//	EX_Trig:BOOL;       // 
	
//	bLayerChanging:BOOL;// 切换成功
//END_VAR    
VAR_IN_OUT
	stfbIJP07         :ST_IJP;
	stItpToPlc :NCTOPLC_NCICHANNEL_REF;
	stPlcToItp:PLCTONC_NCICHANNEL_REF;
END_VAR
VAR
	//HshakeM10Tim:TON;
	//fbGetMFunc:ItpGetHskMFunc;(*获取握手型M函数编号*)	
  //  fbIsMFunc:ItpIsHskMFunc;	(*获取握手型M函数是否触发*)	
    fbConfirm:ItpConfirmHsk;(*复位握手型M函数*)	
  //  fbResetFastMFuncEx:ItpResetFastMFuncEx;
	nActMFuncNr:INT;
	bMFuncEnable: BOOL;
	bMFuncNr:ARRAY[1..159] OF BOOL;
    bQuitMFuncNr:ARRAY[1..159] OF BOOL;
	I: INT;
	EX_Trigtimer:TON;
	EX_TrigHtimer:TON;
    EX_Trigtimertrig:R_TRIG;
	EX_TrigHtimertrig:R_TRIG;
	EX_Trigtime1:TIME;
	EX_Trig:BOOL;       // 
	EX_TrigH:BOOL;       // 
	EX_PringDonetrig:R_TRIG;
	EX_bEl5131_Ftrig:F_TRIG;
	EX_bEl5131_FtrigH:F_TRIG;
END_VAR

nActMFuncNr:=ItpGetHskMFunc(sNCIToPlc:=stItpToPlc);
bMFuncEnable:=ItpIsHskMFunc(sNCIToPlc:=stItpToPlc);
// 
EX_PringDonetrig(CLK:=stfbIJP07.bPrintDone  OR stfbIJP07.bLoadPGMExe, Q=> );
IF  EX_PringDonetrig.Q THEN
		EX_Trig:=FALSE;
		EX_TrigH:=FALSE;
		stfbIJP07.bEx_Trig:=FALSE;
		stfbIJP07.bEx_TrigH:=FALSE;
		stfbIJP07.bEl5131_TrigH:=FALSE;
		stfbIJP07.bEl5131_Trig:=false;
END_IF
// 高压触发
EX_Trigtime1:=INT_TO_TIME(MAX(0,stfbIJP07.iJetOnDelay));
EX_TrigHtimer(IN:=EX_TrigH OR stfbIJP07.bEl5131_TrigH , PT:=EX_Trigtime1,Q=> , ET=> );
IF MAX(0,stfbIJP07.iJetOnDelay) >0 THEN
  EX_TrigHtimertrig(CLK:=EX_TrigHtimer.Q , Q=> );
  IF EX_TrigHtimertrig.Q THEN		
	 stfbIJP07.bEx_TrigH:=TRUE;
  END_IF
ELSE
	EX_TrigHtimertrig(CLK:=EX_TrigH OR stfbIJP07.bEl5131_TrigH , Q=> );
	IF EX_TrigHtimertrig.Q THEN
		stfbIJP07.bEx_TrigH:=TRUE;
	 END_IF
END_IF
// 气压触发
EX_Trigtimertrig(CLK:=EX_Trig OR stfbIJP07.bEl5131_Trig  , Q=> );
IF EX_Trigtimertrig.Q THEN
   stfbIJP07.bEx_Trig:=TRUE;
END_IF
//  比较复位
EX_bEl5131_Ftrig(CLK:= stfbIJP07.bEl5131_Trig, Q=> );
IF EX_bEl5131_Ftrig.Q  THEN
	EX_Trig:=FALSE;
	stfbIJP07.bEx_Trig:=FALSE;
//	stfbIJP07.bEl5131_Trig:=FALSE;
END_IF
EX_bEl5131_FtrigH(CLK:=stfbIJP07.bEl5131_TrigH, Q=> );
IF  EX_bEl5131_FtrigH.Q THEN
	EX_TrigH:=FALSE;
	stfbIJP07.bEx_TrigH:=FALSE;
//	stfbIJP07.bEl5131_TrigH:=FALSE;
END_IF
IF bMFuncEnable THEN
  CASE nActMFuncNr OF 
	 10:(**开触发**)
	    EX_Trig:=TRUE;
        fbConfirm(
         	bExecute:= TRUE, 
	        sNciToPlc:= stItpToPlc, 
	        sPlcToNci:= stPlcToItp, 
	        bBusy=> , 
	        bErr=> , 
	        nErrId=> );
	 11:(**关触发**)
	     EX_Trig:=FALSE;
	     stfbIJP07.bEx_Trig:=FALSE;
        fbConfirm(
         	bExecute:= TRUE, 
	        sNciToPlc:= stItpToPlc, 
	        sPlcToNci:= stPlcToItp, 
	        bBusy=> , 
	        bErr=> , 
	        nErrId=> );
    12:(**打印完成**)
	    stfbIJP07.bPrintDone:=TRUE;
//		EX_Trig:=FALSE;
//		EX_TrigH:=FALSE;
//		stfbIJP07.bEx_Trig:=FALSE;
//		stfbIJP07.bEx_TrigH:=FALSE;
        fbConfirm(
         	bExecute:= TRUE, 
	        sNciToPlc:= stItpToPlc, 
	        sPlcToNci:= stPlcToItp, 
	        bBusy=> , 
	        bErr=> , 
	        nErrId=> );
			
	13:(**图层切换**)
	    stfbIJP07.bLayerChanging:=TRUE;
		IF stfbIJP07.bLayerChanged AND stfbIJP07.bLayerChanging=TRUE THEN			
		 stfbIJP07.bLayerChanging:=FALSE;
		 stfbIJP07.bLayerChanged:=FALSE;
		 fbConfirm(
         	bExecute:= TRUE, 
	        sNciToPlc:= stItpToPlc, 
	        sPlcToNci:= stPlcToItp, 
	        bBusy=> , 
	        bErr=> , 
	        nErrId=> );		
	     END_IF
     20:(** 开高压触发**)
        Ex_TrigH:=TRUE;
        fbConfirm(
         	bExecute:= TRUE, 
	        sNciToPlc:= stItpToPlc, 
	        sPlcToNci:= stPlcToItp, 
	        bBusy=> , 
	        bErr=> , 
	        nErrId=> );
	 21:(** 关高压触发**)
	     EX_TrigH:=FALSE;
		 stfbIJP07.bEx_TrigH:=FALSE;     //触发开关
        fbConfirm(
         	bExecute:= TRUE, 
	        sNciToPlc:= stItpToPlc, 
	        sPlcToNci:= stPlcToItp, 
	        bBusy=> , 
	        bErr=> , 
	        nErrId=> ); 
	
     22: (** 注射泵触发开 **)
        Com_GVLS.stPump.bEX_PumpTrigOn := TRUE;  
        Com_GVLS.stPump.bEX_PumpTrigOff := FALSE;
        fbConfirm(
            bExecute:= TRUE, 
            sNciToPlc:= stItpToPlc, 
            sPlcToNci:= stPlcToItp, 
            bBusy=> , 
            bErr=> , 
            nErrId=> );

     23: (** 注射泵触发关 **)
        Com_GVLS.stPump.bEX_PumpTrigOn := FALSE;  
        Com_GVLS.stPump.bEX_PumpTrigOff := TRUE;
        fbConfirm(
            bExecute:= TRUE, 
            sNciToPlc:= stItpToPlc, 
            sPlcToNci:= stPlcToItp, 
            bBusy=> , 
            bErr=> , 
            nErrId=> );
		
  END_CASE
ELSE
  fbConfirm(bExecute:= FALSE,sNciToPlc:= stItpToPlc,sPlcToNci:= stPlcToItp);
END_IF

END_FUNCTION_BLOCK

// ---- FB/02_NCI/FB/FB_011WriteRParameter.TcPOU
FUNCTION_BLOCK FB_011WriteRParameter

VAR_INPUT
	Execute:BOOL;
	fbnChannelid:UDINT;
	nRParamAry:ARRAY[0..19] OF LREAL;
END_VAR
VAR_OUTPUT
END_VAR
VAR
	fbWriteRParams:ItpWriteRParams;
END_VAR


fbWriteRParams(
	bExecute:= Execute, 
	nChnId:= fbnChannelid, 
	pAddr:= ADR(nRParamAry), 
	nIndex:= 0, 
	nCount:= 10, 
	tTimeOut:= T#2S, 
	bBusy=> , 
	bErr=> , 
	nErrId=> );

END_FUNCTION_BLOCK

// ---- FB/02_NCI/FB/FB_010_ReadRParameter.TcPOU
FUNCTION_BLOCK FB_010_ReadRParameter

VAR_INPUT
	Execute:BOOL;
    fbnChannelid:UDINT;	
END_VAR
VAR_OUTPUT
	nRParamAry:ARRAY[0..19] OF LREAL;
END_VAR
VAR
	fbReadRParams:ItpReadRParams;
END_VAR



	fbReadRParams(
	bExecute:= Execute, 
	nChnId:= fbnChannelid, 
	pAddr:= ADR(nRParamAry), 
	nIndex:= 0, 
	nCount:= 20, 
	tTimeOut:= T#2S, 
	bBusy=> , 
	bErr=> , 
	nErrId=> );

END_FUNCTION_BLOCK

// ---- FB/02_NCI/FB/FB_013_WriteZeroShiftEx.TcPOU
FUNCTION_BLOCK FB_013_WriteZeroShiftEx
VAR_INPUT
	bExecute:BOOL;
	nZsNo:UDINT;
	tTimeOut:TIME;
	lZeroShiftX             :LREAL                      ;           //X偏移值
	lZeroShiftY             :LREAL                      ;           //Y偏移值
	lZeroShiftZ             :LREAL                      ;           //Z偏移值	
END_VAR
VAR_OUTPUT
	bBusy:BOOL;
	bErr:BOOL;
	nErrId:UDINT;
END_VAR
VAR_IN_OUT
	stItpToPlc :NCTOPLC_NCICHANNEL_REF;
END_VAR
VAR
stZerohiftDesc:ZeroShiftDesc;
fbWriteZeroShiftEx:ItpWriteZeroShiftEx;
END_VAR

fbWriteZeroShiftEx(bExecute:=bExecute,nZsNo:=nZsNo,tTimeOut:=tTimeOut,sNciToPlc:=stItpToPlc,sZeroShiftDesc:=stZerohiftDesc,bBusy=>bBusy,bErr=>bErr,nErrId=>nErrId);
stZerohiftDesc.fShiftX:=lZeroShiftX;
stZerohiftDesc.fShiftY:=lZeroShiftY;
stZerohiftDesc.fShiftZ:=lZeroShiftZ;

END_FUNCTION_BLOCK

// ---- POUs/3_Aio/AIO.TcPOU
PROGRAM AIO
VAR
	fbAdc:ARRAY[1..2,1..4] OF FB_ADC;	
	fbDac:ARRAY[1..2,1..4] OF FB_DAC;
	ro2:REAL;
	ro3:REAL;
END_VAR

(*ACT*)
AD();
DA();

ACTION AD:
(*A-D*)	
(**)
//底部负压显示表  0   -101kap
fbAdc[1,1]
    (
	rAnalogIn:=        AX_1[1] , 
	rAnalogLowLMT:=    REAL#0 , 
	rAanlogUpperLMT:=  REAL#16000, 
	rAnalogRef1:=      REAL#14870, 
	rDigitalRef1:=     REAL#-90, 
	rAnalogRef2:=      REAL#6850, 
	rDigitalRef2:=     REAL#-27.7, 
	rDigitalOut=>      stAIO.rAI1 , 
    );
//针头正负压显示表   -0.1  1.0Mpa
fbAdc[1,2]
    (
	rAnalogIn:=        AX_1[2] , 
	rAnalogLowLMT:=    REAL#10 , 
	rAanlogUpperLMT:=  REAL#32700, 
	rAnalogRef1:=      REAL#4541, 
	rDigitalRef1:=     REAL#97, 
	rAnalogRef2:=      REAL#3896, 
	rDigitalRef2:=     REAL#47, 
	rDigitalOut=>      stAIO.rAI2 , 
    );

(*
//针头负压比例阀反馈	
fbAdc[2,2]
    (
	rAnalogIn:=        AX_2[2] , 
	rAnalogLowLMT:=    REAL#10 , 
	rAanlogUpperLMT:=  REAL#32700, 
	rAnalogRef1:=      REAL#3384, 
	rDigitalRef1:=     REAL#0, 
	rAnalogRef2:=      REAL#6345, 
	rDigitalRef2:=     REAL#-20, 
	rDigitalOut=>      stAIO.rAI6 , 
    );	
//针头正压比例阀反馈
fbAdc[2,3]
    (
	rAnalogIn:=        AX_2[3] , 
	rAnalogLowLMT:=    REAL#0 , 
	rAanlogUpperLMT:=  REAL#32700, 
	rAnalogRef1:=      REAL#2368, 
	rDigitalRef1:=     REAL#200, 
	rAnalogRef2:=      REAL#1716, 
	rDigitalRef2:=     REAL#150, 
	rDigitalOut=>      stAIO.rAI7 , 
    );	
*)
END_ACTION

ACTION DA:
(*D-A*)	
//针头正压比例阀 ITV0090-3BL -1--100kpa
IF NOT stIJP.bEx_Trig AND  NOT stIJP.bEx_TrigH THEN
	ro2:= stAIO.rAO2;
ELSE
	ro2:= 0	;
END_IF
fbDac[1,2]
    (
	rDigitalIn:=     ro2 , 
	rAnalogLowLMT:=   REAL#0, 
	rAanlogUpperLMT:= REAL#32767, 
	rAnalogRef1:=     REAL#6149, 
	rDigitalRef1:=    REAL#-15 , 
	rAnalogRef2:=     REAL#9951, 
	rDigitalRef2:=    REAL#-27, 
	rAnalogOut=>      AY_1[2] , 
    );

//AY_1[2]:=0;
//针头正压比例阀  ITV-0030-3BL  0.001-0.5MPA 1-500kpa
IF stIJP.bEx_Trig AND  stIJP.bEx_TrigH THEN
	ro3:= stAIO.rAO3;
ELSE
	ro3:= 0	;
END_IF
fbDac[1,3]
    (
	rDigitalIn:=      ro3, 
	rAnalogLowLMT:=   REAL#0 , 
	rAanlogUpperLMT:= REAL#32767, 
	rAnalogRef1:=     REAL#3031, 
	rDigitalRef1:=    REAL#46 , 
	rAnalogRef2:=     REAL#10193, 
	rDigitalRef2:=    REAL#154, 
	rAnalogOut=>      AY_1[3] , 
    );
END_ACTION

END_PROGRAM

// ---- FB/11_AIO/FB/FB_ADC.TcPOU
FUNCTION_BLOCK FB_ADC
VAR
	bFirstRun    :BOOL := TRUE;
	rAnaIn       :REAL;
END_VAR
VAR_INPUT
	rAnalogIn			:			INT	;		     //模拟量输入      显示表/比例阀反馈
	rAnalogLowLMT		:			REAL	;		 //模拟量下限值     0
	rAanlogUpperLMT		:			REAL	;	     //模拟量上限值     32767     
	rAnalogRef1			:			REAL	;		 //参考点1：       模拟量 例10
	rDigitalRef1		:			REAL	;		 //参考点1：       数字量 例0.1kpa
	rAnalogRef2			:			REAL	;		 //参考点2：       模拟量  例5000
	rDigitalRef2		:			REAL	;		 //参考点2：       数字量  例0.3kpa
END_VAR
VAR_OUTPUT
	rDigitalOut			:			REAL	;		 //数字量显示      上位机显示
	bError				:			BOOL	;		 //错误
END_VAR

IF bFirstRun THEN
	IF ABS(rAnalogLowLMT) < 0.001 THEN
		rAnalogLowLMT := -50000.0;
	END_IF;
	IF ABS(rAanlogUpperLMT) < 0.001 THEN
		rAanlogUpperLMT := 50000.0;
	END_IF;
END_IF;
bFirstRun := FALSE;

rAnaIn    :=LIMIT(rAnalogLowLMT, rAnalogIn, rAanlogUpperLMT);

IF 	ABS(rDigitalRef2 - rDigitalRef1) > 0.00001 AND ABS(rAnalogRef2 - rAnalogRef1) > 0.00001 THEN
	rDigitalOut := (rAnaIn - rAnalogRef1) * (rDigitalRef2 - rDigitalRef1)/(rAnalogRef2 - rAnalogRef1)+ rDigitalRef1;	
	bError := FALSE;
ELSE
	rDigitalOut := 0;
	bError := TRUE;
END_IF;

END_FUNCTION_BLOCK

// ---- FB/11_AIO/FB/FB_DAC.TcPOU
FUNCTION_BLOCK FB_DAC

VAR
	rAnaOut         :REAL;
	bFirstRun: BOOL := TRUE;
END_VAR
VAR_INPUT
	rDigitalIn			:			REAL	;		//数字量输入     例上位机
	rAnalogLowLMT		:			REAL	;		//模拟量下限     0
	rAanlogUpperLMT		:			REAL	;		//模拟量上限     32767
	rAnalogRef1			:			REAL	;		//参考点1：模拟量
	rDigitalRef1		:			REAL	;		//参考点1：数字量
	rAnalogRef2			:			REAL	;		//参考点2：模拟量
	rDigitalRef2		:			REAL	;		//参考点2：数字量
END_VAR
VAR_OUTPUT
	rAnalogOut			:			INT	    ;		//模拟量输出
	bError				:			BOOL	;		//错误
END_VAR

IF bFirstRun THEN
	IF ABS(rAnalogLowLMT) < 0.01 THEN
		rAanlogUpperLMT := -50000.0;
	END_IF;
	IF ABS(rAanlogUpperLMT) < 0.01 THEN
		rAanlogUpperLMT := 50000.0;
	END_IF;
END_IF;
bFirstRun:=FALSE;
IF rDigitalIn<>0 THEN
IF ABS(rAnalogRef2 - rAnalogRef1) > 0.00001 AND ABS(rDigitalRef2 - rDigitalRef1) >0.00001 THEN
	rAnaOut:=(rDigitalIn - rDigitalRef1) * (rAnalogRef2 - rAnalogRef1)/(rDigitalRef2 -rDigitalRef1) +rAnalogRef1;
	rAnaOut:=LIMIT(rAnalogLowLMT,rAnaOut,rAanlogUpperLMT);
	rAnalogOut:=REAL_TO_INT(rAnaOut);
	bError:=FALSE;
ELSE
	rAnalogOut := 0;
	bError     := TRUE;
END_IF;	
ELSE
rAnalogOut := 0;
END_IF;

END_FUNCTION_BLOCK

// ---- POUs/System_State.TcPOU
PROGRAM System_State
VAR
	udiError: INT;
	NCI_BII_IOLINK: INT;
	biXLIMP: INT;
	HomeStep:INT;
	HomTime:ton;
	bPowerOK: INT;
	SysHomstep:INT;
	SysHomstept:ton;
	SysHomTrig:R_trig;	
	Setposition :TON;
	fbReadNetid:FB_ReadNetid;
	posEdgEmg:r_trig;
END_VAR

//(* 整机首次上点延时*)
tonSystemFirstRun(IN:=TRUE , PT:= T#10S);
posEdgeFirstRun(CLK:=tonSystemFirstRun.Q , Q=> );
IF posEdgeFirstRun.Q THEN
   fbReadNetid(sNetID=>stSystem.strNetID);
END_IF
(*1-*EMS*)
stSystem.arErrorID[15]:=NOT X000001;
(*2-*Reset*)
IF stSystem.bReset THEN
   arstAxis[1].Control.bReset_A:=TRUE;
   arstAxis[2].Control.bReset_A:=TRUE;
   arstAxis[3].Control.bReset_A:=TRUE;
   arstAxis[4].Control.bReset_A:=TRUE;
   arstAxis[5].Control.bReset_A:=TRUE;
   arstAxis[6].Control.bReset_A:=TRUE;
   arstAxis[7].Control.bReset_A:=TRUE;
   arstAxis[8].Control.bReset_A:=TRUE;
   arstAxis[9].Control.bReset_A:=TRUE;
   arstAxis[10].Control.bReset_A:=TRUE;
   stSystem.bReset:=FALSE;
END_IF
(*3-*Stop*)
IF stSystem.bStop THEN
   arstAxis[1].Control.bStop_A:=TRUE;
   arstAxis[2].Control.bStop_A:=TRUE;
   arstAxis[3].Control.bStop_A:=TRUE;
   arstAxis[4].Control.bStop_A:=TRUE;
   arstAxis[5].Control.bStop_A:=TRUE;
   arstAxis[6].Control.bStop_A:=TRUE;
   arstAxis[7].Control.bStop_A:=TRUE;
   arstAxis[8].Control.bStop_A:=TRUE;
   arstAxis[9].Control.bStop_A:=TRUE;
   arstAxis[10].Control.bStop_A:=TRUE;
   stSystem.bStop:=FALSE;
END_IF
(*4-*Axis_Power*)
IF stSystem.bPower AND NOT stSystem.arErrorID[15] THEN
   arstAxis[1].Control.bPowerOn:=TRUE;
   arstAxis[2].Control.bPowerOn:=TRUE;
   arstAxis[3].Control.bPowerOn:=TRUE;
   arstAxis[4].Control.bPowerOn:=TRUE;
   arstAxis[5].Control.bPowerOn:=TRUE;
   arstAxis[6].Control.bPowerOn:=TRUE;
   arstAxis[7].Control.bPowerOn:=TRUE;
   arstAxis[8].Control.bPowerOn:=TRUE;
   arstAxis[9].Control.bPowerOn:=TRUE;
   arstAxis[10].Control.bPowerOn:=TRUE;
//   stSystem.bStop:=FALSE;
END_IF
posEdgEmg(CLK:=stSystem.arErrorID[15] , Q=> );
IF posEdgEmg.Q THEN
   arstAxis[1].Control.bPowerOn:=FALSE;
   arstAxis[2].Control.bPowerOn:=FALSE;
   arstAxis[3].Control.bPowerOn:=FALSE;
   arstAxis[4].Control.bPowerOn:=FALSE;
   arstAxis[5].Control.bPowerOn:=FALSE;
   arstAxis[6].Control.bPowerOn:=FALSE;
   arstAxis[7].Control.bPowerOn:=FALSE;
   arstAxis[8].Control.bPowerOn:=FALSE;
   arstAxis[9].Control.bPowerOn:=FALSE;
   arstAxis[10].Control.bPowerOn:=FALSE;
END_IF

(*5-*ALL_Power*)
stSystem.bPowerOK:=arstAxis[1].State.bPowerOK AND arstAxis[2].State.bPowerOK AND arstAxis[3].State.bPowerOK AND arstAxis[4].State.bPowerOK AND arstAxis[5].State.bPowerOK	AND arstAxis[6].State.bPowerOK;
(*6-*Home*)
SysHomTrig(CLK:=stSystem.bHOME AND stSystem.bPowerOK , Q=> );
IF SysHomTrig.Q THEN
	HOMEstep:=0;
	SysHomstep:=5;
END_IF
CASE SysHomstep OF
	5: 
       Axis_Home();
	   SysHomstept(in:=TRUE,pt:=T#20MS);
	   IF stSystem.bHOMEOK AND SysHomstept.Q THEN
		 SysHomstept(in:=FALSE);
         stSystem.bHOME:=FALSE;  
		 SysHomstep:=10;  	   
	   END_IF
END_CASE


Y000007:=arstVac[1].bVacuumReq;
Y000006:=NOT	arstVac[1].bVacuumReq;

Y000009:=arstVac[2].bVacuumReq;
Y000008:=NOT	arstVac[2].bVacuumReq;

Y000010:=arstVac[3].bVacuumReq;
Y000011:=NOT	arstVac[3].bVacuumReq;

ACTION Axis_Home:

CASE HOMEstep OF
  0:(*  *) 
      stSystem.bHOMEOK := FALSE;  
      arstAxis[1].Control.bHome_A:=FALSE;
	  arstAxis[2].Control.bHome_A:=FALSE; 
	  arstAxis[3].Control.bHome_A:=FALSE;
	  arstAxis[4].Control.bHome_A:=FALSE;
	  
      arstAxis[5].Control.bHome_A:=FALSE;
	  arstAxis[6].Control.bHome_A:=FALSE;
	  arstAxis[7].Control.bHome_A:=FALSE;
	  arstAxis[8].Control.bHome_A:=FALSE;
	  arstAxis[9].Control.bHome_A:=FALSE;
	  arstAxis[10].Control.bHome_A:=FALSE;
	  stSystem.bHoming:=TRUE;
	  HOMEstep:=5;
  5: // 绝对值轴回零
      arstAxis[6].Control.bHome_A:=TRUE;
	  arstAxis[7].Control.bHome_A:=TRUE;
	  arstAxis[8].Control.bHome_A:=TRUE;
	  arstAxis[9].Control.bHome_A:=TRUE;
	  arstAxis[10].Control.bHome_A:=TRUE;
	  HOMEstep:=10;
  10:(*Z轴回零动作 Z1 Z2*)
     arstAxis[4].Control.bHome_A:=TRUE;
	 arstAxis[5].Control.bHome_A:=TRUE;
	 HomeStep:=15;
  15:	
	 HomTIME(IN:=TRUE,PT:=T#20MS,Q=>,ET=>);
	 IF arstAxis[4].State.bHome_OK AND NOT arstAxis[4].State.bHoming AND 
        arstAxis[5].State.bHome_OK AND NOT arstAxis[5].State.bHoming AND HomTIME.Q THEN
		HomTIME(IN:=FALSE);
		HomeStep:=20;
	 ELSIF arstAxis[4].State.bError   AND  arstAxis[5].State.bError  AND HomTIME.Q THEN
		HomTIME(IN:=FALSE);
		HomeStep:=1000;
	 END_IF
	   
  20:(* R回零动作*)
     arstAxis[3].Control.bHome_A:=TRUE;
	 HomTIME(IN:=TRUE,PT:=T#20MS,Q=>,ET=>);
	 IF arstAxis[3].State.bHome_OK AND NOT arstAxis[3].State.bHoming AND HomTIME.Q   THEN
		HomTIME(IN:=FALSE);
		HomeStep:=30;
	 ELSIF arstAxis[3].State.bError   AND HomTIME.Q THEN
		HomTIME(IN:=FALSE);
		HomeStep:=1000;
	 END_IF
	 
  30:(* XY回零动作*)
     arstAxis[1].Control.bHome_A:=TRUE;
	 arstAxis[2].Control.bHome_A:=TRUE;
		HomeStep:=35;
35:
     HomTIME(IN:=TRUE,PT:=T#20MS,Q=>,ET=>);
  	 IF arstAxis[1].State.bHome_OK  AND arstAxis[2].State.bHome_OK AND HomTIME.Q THEN
		HomTIME(IN:=FALSE);
		HomeStep:=40;
	 ELSIF arstAxis[1].State.bError   AND  arstAxis[2].State.bError  AND HomTIME.Q THEN
		HomTIME(IN:=FALSE);
		HomeStep:=1000;
	 END_IF 
  40:(* xy位置比较写入参考位置设置*)	
//     arstCamCtrlIO[1].bSetRefPos:=TRUE;
//	 arstCamCtrlIO[2].bSetRefPos:=TRUE;
//	 Setposition(IN:=arstCamCtrlIO[1].bSetRefPos AND stCamCtrlIO[2].bSetRefPos ,PT:=T#20MS,Q=>,ET=>);
//	 IF Setposition.Q THEN
		HomeStep:=50; 
//	 END_IF
	 
  50:(* 重新使能 *) 
//     stCamCtrlIO[1].bSetRefPos:=FALSE;
//	 stCamCtrlIO[2].bSetRefPos:=FALSE;
//	 IF stCamCtrlIO[1].bSetRefPos=FALSE AND  stCamCtrlIO[2].bSetRefPos=FALSE THEN
	 HOMEstep:=60;
//	 END_IF
	 
  60:(*建立NCI通道*)
     stSystem.bHoming:=FALSE;
     stSystem.bHOMEOK:=TRUE;
 1000:
     stSystem.bHoming:=FALSE;
     stSystem.bHOMEOK:=FALSE;				
END_CASE
END_ACTION

END_PROGRAM

// ---- FB/51_Netid/FB_ReadNetid.TcPOU
FUNCTION_BLOCK FB_ReadNetid
VAR_INPUT

END_VAR
VAR_OUTPUT
	sNetID:STRING;
END_VAR
VAR
    tAmsNetid AT %I*  :AmsNetId;  
    i:INT;  
END_VAR

// 将6个字节转换为点分格式
sNetID := BYTE_TO_STRING(tAmsNetid[0]);
FOR i := 1 TO 5 DO
    sNetID := CONCAT(CONCAT(sNetID, '.'), BYTE_TO_STRING(tAmsNetid[i]));
END_FOR

END_FUNCTION_BLOCK

// ---- POUs/07_PDMctr/PDMctr.TcPOU
PROGRAM PDMctr
VAR
	FB_PDMSCtr:FB_PDMSCtr;

	TonWrite: TON;
	TonWriteQ: BOOL;

END_VAR

FB_PDMSCtr(
	stLightCtr:= stLightCtr, 
	strNetID:=stSystem.strNetID , 
	uiSlaveAddr:=1010, 
	wIndex:= 16#8000, 
	wstrCommPara=> );

END_PROGRAM

// ---- FB/31_PDMSCtr/FB/FB_PDMSCtr.TcPOU
// 主功能块定义：PDMS光源控制器
FUNCTION_BLOCK FB_PDMSCtr
// 输入输出参数：灯光控制结构体（双向传递）
VAR_IN_OUT
    stLightCtr: ST_LightCtr;  // 4个通道亮度的设定值和实际亮度值
END_VAR

VAR_INPUT
	  // EtherCAT模块网络标识（设备地址）
    strNetID: STRING;     // 模块的NetID地址字符串
    // 模块从站地址（设备编号）
    uiSlaveAddr: UINT;    // 从站地址（无符号整数）
    // COM口功能索引号（对象字典索引）
    wIndex: WORD;         // CoE通信索引号（字类型）
//	// 通讯参数设置触发，上升沿有效
//	bCommParaSetExe: BOOL;
//	// 波特率设定，默认设定7-19200。
//	// 对应关系：1-300；2-600；3-1200；4-2400；5-4800；6-9600；7-19200；8-38400；9-57600；10-115200
//	siBaudrateSet: SINT := 7;
//	// 传输格式设定， 默认设定3-8N1。
//	// 对应关系：1-7E1；2-7O1；3-8N1；4-8E1；5-8O1；8-7N2；9-7E2；10-7O2；11-8N2；12-8E2；13-8O2。
//	siDataFrameSet: SINT := 3;
//	// RTS/CTS功能设定。默认设定0 - 关闭。
//	// 对应关系：0-关闭；1-打开。
//	siRTSCTSStateSet: SINT := 0;
END_VAR
// 输出参数：通信状态信息
VAR_OUTPUT
    // 当前端口通讯参数描述（宽字符串输出）
    wstrCommPara: WSTRING;  // 显示波特率、数据格式等通信参数
END_VAR

// 局部变量声明区域
VAR
    // 运行状态标志
    bFirstRun: BOOL;        // 首次运行标志（TRUE表示第一次运行）
    Ton0: TON;              // 初始化定时器（用于首次运行延时）
    TonWrite: TON;          // 数据写入定时器（控制发送时序）
    TonWriteQ:BOOL;         // 写入定时器状态标志
    bFirstTrig: BOOL;       // 首次触发标志（用于初始化操作）
    
    // 定时闪烁功能块（生成周期脉冲）
    fbBlink1s: BLINK;       // 1秒闪烁器（用于周期触发读取操作）
   
    // 变化检测功能块
    rtrigChanIntensityChg: R_TRIG;      // 上升沿检测器（检测亮度变化）
    
    // 通信时序控制定时器
    Ton10: TON;             // 10ms定时器（用于步骤10的超时控制）
    Ton20: TON;             // 20ms定时器（用于步骤20的超时控制）
    
    // 状态机控制变量
    iStep: INT := 100;      // 状态机步骤计数器（初始值100）
    
    // 数据帧缓冲区
    arSendData: ARRAY[0..16] OF BYTE := [16#40, 16#0E ,16#01, 16#0, 16#1A, 16#0, 0, 16#1A, 16#1, 0, 16#1A, 16#2, 0, 16#1A, 16#3, 0, 0];  // 设置命令数据帧
    fbSendData: SendData;   // 数据发送功能块实例
    
    // 读取命令数据帧 
    fbSendData2: SendData;  // 读取数据发送功能块实例
    arSendData2: ARRAY[0..6] OF BYTE := [16#40, 16#4, 16#1, 16#0, 16#31, 16#FF, 16#75];  // 读取命令数据帧
    
    // 数据帧起始和结束标志
    byStart: BYTE := 16#40;  // 数据帧起始字节（0x40）
    byEnd: BYTE := 16#B9;    // 数据帧结束字节（0xB9）
    
    // 接收数据缓冲区
    arReceiveData: ARRAY[0..16] OF BYTE;  // 接收数据存储数组
    fbReceiveData: ReceiveData;           // 数据接收功能块实例
    
    // 串口通信控制功能块
    fbSerialLineControl: SerialLineControl;  // 串行线路控制功能块
    
    // 硬件映射（连接到实际的I/O模块）
    COMin_MASTER AT %I*: EL6inData22B;    // 主站输入数据缓冲区（映射到实际输入地址）
    COMout_MASTER AT %Q*: EL6outData22B;  // 主站输出数据缓冲区（映射到实际输出地址）
    
    // 通信缓冲区
    RxBuffer_MASTER: ComBuffer;  // 接收缓冲区（存储接收到的数据）
    TxBuffer_MASTER: ComBuffer;  // 发送缓冲区（存储要发送的数据）
    
    // 亮度变化执行标志
    bChanIntensityChgExe: BOOL;  // 通道亮度变化执行标志（TRUE需要更新亮度）
    
    // 校验码计算变量
    crc:UINT;    // 校验和计算变量（无符号整数）
    i:UINT;      // 循环计数器（用于校验计算）
    arReceiveDatatemp:UINT;  // 接收数据临时变量
	
	 
    // CoE通信功能块（用于读取串口参数）
    fbCoEReadBaudrate: FB_EcCoESdoRead;     // 读取波特率功能块
    fbCoEReadDataFrame: FB_EcCoESdoRead;    // 读取数据格式功能块
    fbCoEReadRTSCTSState: FB_EcCoESdoRead;  // 读取流控状态功能块
    
    // CoE通信功能块（用于设置串口参数）
    fbCoEWriteBaudrate: FB_EcCoESdoWrite;    // 写入波特率功能块
    fbCoEWriteDataFrame: FB_EcCoESdoWrite;   // 写入数据格式功能块
    fbCoeWriteRTSCTSState: FB_EcCoESdoWrite; // 写入流控状态功能块
    
    // 临时变量用于存储读取的通信参数
    siBaudrateReadTemp: SINT;           // 临时存储读取的波特率值
    wstrBaudrateRead: WSTRING;          // 波特率描述字符串
    siDataFrameReadTemp: SINT;          // 临时存储读取的数据格式值
    wstrDataFrameRead: WSTRING;         // 数据格式描述字符串
    siRTSCTSStateReadTemp: SINT;        // 临时存储读取的流控状态值
    wstrRTSCTSStateRead: WSTRING;       // 流控状态描述字符串
    wstrCommParaTemp: WSTRING;          // 临时通信参数字符串
    
    
END_VAR

(****
		使用串口控制模块-EL6002控制Wordop-PDMS-4输出紧凑型光源控制器
		
		2024-1-4  1-设置并输出通讯速率/格式更换
							2-设置四通道光源亮度参数，并读出
							3-判定设定值与当前值不同，自动更改
***)
// 首次运行初始化处理
IF bFirstRun THEN
    bFirstTrig := TRUE;          // 设置首次触发标志为TRUE
    Ton0(IN := bFirstRun, PT := TIME#10MS, Q => , ET => );  // 启动10ms定时器
    IF Ton0.Q THEN               // 如果定时器到时 
        bFirstTrig := FALSE;     // 清除首次触发标志
        bFirstRun := FALSE;      // 清除首次运行标志（后续不再进入此分支）
    END_IF    
END_IF

(*
{region"通讯参数设定"}
//通讯速率、通讯格式读取
fbBlink1s(ENABLE:=TRUE , TIMELOW:=TIME#1S , TIMEHIGH:=TIME#1S , OUT=> );

fbCoEReadBaudrate(
	sNetId:=strNetID , 
	nSlaveAddr:=uiSlaveAddr , 
	nSubIndex:=16#11 , 
	nIndex:=wIndex , 
	pDstBuf:=ADR(siBaudrateReadTemp) , 
	cbBufLen:=SIZEOF(siBaudrateReadTemp) , 
	bExecute:=fbBlink1s.OUT , 
	tTimeout:= , 
	bBusy=> , 
	bError=> , 
	nErrId=> , 
	cbRead=> );
	
fbCoEReadDataFrame(
	sNetId:=strNetID , 
	nSlaveAddr:=uiSlaveAddr , 
	nSubIndex:= 16#15, 
	nIndex:= wIndex, 
	pDstBuf:=ADR(siDataFrameReadTemp)  , 
	cbBufLen:=SIZEOF(siDataFrameReadTemp) , 
	bExecute:=fbBlink1s.OUT , 
	tTimeout:= , 
	bBusy=> , 
	bError=> , 
	nErrId=> , 
	cbRead=> );

fbCoEReadRTSCTSState(
	sNetId:=strNetID , 
	nSlaveAddr:=uiSlaveAddr , 
	nSubIndex:=16#01 , 
	nIndex:=wIndex , 
	pDstBuf:= ADR(siRTSCTSStateReadTemp), 
	cbBufLen:=SIZEOF(siRTSCTSStateReadTemp) , 
	bExecute:=fbBlink1s.OUT , 
	tTimeout:= , 
	bBusy=> , 
	bError=> , 
	nErrId=> , 
	cbRead=> );
	
CASE siBaudrateReadTemp OF 
	1:
		wstrBaudrateRead := "当前波特率：300，";
	2:
		wstrBaudrateRead := "当前波特率：600，";
	3:
		wstrBaudrateRead := "当前波特率：1200，";
	4:
		wstrBaudrateRead := "当前波特率：2400，";
	5:
		wstrBaudrateRead := "当前波特率：4800，";
	6:
		wstrBaudrateRead := "当前波特率：9600，";
	7:
		wstrBaudrateRead := "当前波特率：19200，";
	8:
		wstrBaudrateRead := "当前波特率：38400，";
	9:
		wstrBaudrateRead := "当前波特率：57600，";
	10:
		wstrBaudrateRead := "当前波特率：115200，";	
END_CASE

CASE siDataFrameReadTemp OF 
	1:
		wstrDataFrameRead:= "当前传输格式：7E1，数据位7，停止位1，偶校验，";
	2:
		wstrDataFrameRead:= "当前传输格式：7O1，数据位7，停止位1，奇校验，"	;
	3:
		wstrDataFrameRead:= "当前传输格式：8N1，数据位8，停止位1，无校验，"	;
	4:
		wstrDataFrameRead:= "当前传输格式：8E1，数据位8，停止位1，偶校验，"	;
	5:
		wstrDataFrameRead:= "当前传输格式：8O1，数据位8，停止位1，奇校验，"	;
	8:
		wstrDataFrameRead:= "当前传输格式：7N2，数据位7，停止位2，无校验，"	;
	9:
		wstrDataFrameRead:= "当前传输格式：7E2，数据位7，停止位2，偶校验，"	;
	10:
		wstrDataFrameRead:= "当前传输格式：7O2，数据位7，停止位2，奇校验，"	;
	11:
		wstrDataFrameRead:= "当前传输格式：8N2，数据位8，停止位2，无校验，"	;
	12:
		wstrDataFrameRead:= "当前传输格式：8E2，数据位8，停止位2，偶校验，"	;
	13:
		wstrDataFrameRead:= "当前传输格式：8O2，数据位8，停止位2，奇校验，"	;
	
END_CASE;

CASE siRTSCTSStateReadTemp OF 
	0:
		wstrRTSCTSStateRead:="串口流控未开启";
	1:
		wstrRTSCTSStateRead:="串口流控已开启";	
END_CASE;

wstrCommParaTemp := WCONCAT(STR1:=wstrBaudrateRead,STR2:=wstrDataFrameRead);
wstrCommPara:=WCONCAT(STR1:=wstrCommParaTemp,STR2:=wstrRTSCTSStateRead);
//通讯速率、通讯格式更改

fbCoEWriteBaudrate(
	sNetId:=strNetID , 
	nSlaveAddr:=uiSlaveAddr, 
	nSubIndex:=16#11 , 
	nIndex:=wIndex , 
	pSrcBuf:=ADR(siBaudrateSet) , 
	cbBufLen:=SIZEOF(siBaudrateSet) , 
	bExecute:=bCommParaSetExe OR bFirstTrig, 
	tTimeout:= , 
	bBusy=> , 
	bError=> , 
	nErrId=> );

fbCoEWriteDataFrame(
	sNetId:=strNetID , 
	nSlaveAddr:=uiSlaveAddr , 
	nSubIndex:=16#15 , 
	nIndex:=wIndex , 
	pSrcBuf:=ADR(siDataFrameSet) , 
	cbBufLen:=SIZEOF(siDataFrameSet) , 
	bExecute:=bCommParaSetExe OR bFirstTrig, 
	tTimeout:= , 
	bBusy=> , 
	bError=> , 
	nErrId=> );

fbCoeWriteRTSCTSState(
	sNetId:=strNetID  , 
	nSlaveAddr:=uiSlaveAddr , 
	nSubIndex:=16#01 , 
	nIndex:=wIndex , 
	pSrcBuf:=ADR(siRTSCTSStateSet)  , 
	cbBufLen:= SIZEOF(siRTSCTSStateSet), 
	bExecute:=bCommParaSetExe OR bFirstTrig , 
	tTimeout:= , 
	bBusy=> , 
	bError=> , 
	nErrId=> );
		 
{endregion}
*)	 

{region"通道光源值写入与读取"}	 
//写入值判定
// 通道1亮度值范围限制（保护逻辑）
IF stLightCtr.iChannel1ValueSet < 0 THEN          // 如果设定值小于0
    stLightCtr.iChannel1ValueSet := 0;            // 强制设为最小值0
ELSIF stLightCtr.iChannel1ValueSet > 255 THEN    // 如果设定值大于
    stLightCtr.iChannel1ValueSet := 255;          // 强制设为最大值
END_IF;
	 
// 通道2亮度值范围限制
IF stLightCtr.iChannel2ValueSet < 0 THEN          // 如果设定值小于0
    stLightCtr.iChannel2ValueSet := 0;            // 强制设为最小值0
ELSIF stLightCtr.iChannel2ValueSet > 255 THEN    // 如果设定值大于
    stLightCtr.iChannel2ValueSet := 255;          // 强制设为最大值
END_IF;
	 
// 通道3亮度值范围限制
IF stLightCtr.iChannel3ValueSet < 0 THEN          // 如果设定值小于0
    stLightCtr.iChannel3ValueSet := 0;            // 强制设为最小值0
ELSIF stLightCtr.iChannel3ValueSet > 255 THEN    // 如果设定值大于
    stLightCtr.iChannel3ValueSet := 255;          // 强制设为最大值
END_IF;

// 通道4亮度值范围限制
IF stLightCtr.iChannel4ValueSet < 0 THEN          // 如果设定值小于0
    stLightCtr.iChannel4ValueSet := 0;            // 强制设为最小值0
ELSIF stLightCtr.iChannel4ValueSet > 255 THEN    // 如果设定值大于
    stLightCtr.iChannel4ValueSet := 255;          // 强制设为最大值
END_IF;

//通道参数值写入传输数组中	 
// 将通道1亮度值写入发送数据帧（16位值拆分为2个字节）
//arSendData[6] := UINT_TO_BYTE(SHR(stLightCtr.iChannel1ValueSet, 8));  // 高8位（右移8位取高字节）
arSendData[6] := UINT_TO_BYTE(stLightCtr.iChannel1ValueSet);          // 低8位（直接转换取低字节）
	 
// 将通道2亮度值写入发送数据帧
//arSendData[10] := UINT_TO_BYTE(SHR(stLightCtr.iChannel2ValueSet, 8));  // 高8位
arSendData[9] := UINT_TO_BYTE(stLightCtr.iChannel2ValueSet);          // 低8位
	 
// 将通道3亮度值写入发送数据帧
// arSendData[14] := UINT_TO_BYTE(SHR(stLightCtr.iChannel3ValueSet, 8));  // 高8位
arSendData[12] := UINT_TO_BYTE(stLightCtr.iChannel3ValueSet);          // 低8位
	 
// 将通道4亮度值写入发送数据帧
// arSendData[18] := UINT_TO_BYTE(SHR(stLightCtr.iChannel4ValueSet, 8));  // 高8位
arSendData[15] := UINT_TO_BYTE(stLightCtr.iChannel4ValueSet);          // 低8位 
	 
//校验码计算
//arSendData[20]:=(16#FF AND (16#BD +arSendData[6]+arSendData[7]+arSendData[10]+arSendData[11]
//                            +arSendData[14]+arSendData[15] +arSendData[18]+arSendData[19]));
	 
		  
// 计算数据帧校验码（累加和校验）
crc := 0;                            // 初始化校验和为0
FOR i := 0 TO 15 BY 1 DO             //  循环遍历前16个字节（0-15）
    crc := arSendData[i] + crc;      // 累加每个字节的值
END_FOR
// 取累加和的低8位作为校验码，放入数据帧最后一个位置
arSendData[16] := UINT_TO_BYTE(crc AND 16#FF);  // 与0xFF进行与操作取低8位
	 
		  
//任一通道值改变触发通讯
//TonWrite(IN:=NOT TonWrite.Q , PT:=TIME#200MS , Q=> , ET=> );
//IF TonWrite.Q THEN
	 
// 检测是否需要更新亮度（比较设定值与实际值）
IF stLightCtr.iChannel1ValueSet <> stLightCtr.iChannel1ActValue  // 通道1值变化
    OR stLightCtr.iChannel2ValueSet <> stLightCtr.iChannel2ActValue  // 通道2值变化
    OR stLightCtr.iChannel3ValueSet <> stLightCtr.iChannel3ActValue  // 通道3值变化
    OR stLightCtr.iChannel4ValueSet <> stLightCtr.iChannel4ActValue THEN  // 通道4值变化
    // 如果有任何一个通道的值发生变化
    bChanIntensityChgExe := TRUE;  // 设置亮度变化执行标志为TRUE（需要更新）
 
// 如果所有通道的设定值都与实际值匹配
ELSIF stLightCtr.iChannel1ValueSet = stLightCtr.iChannel1ActValue  // 通道1值匹配
    AND stLightCtr.iChannel2ValueSet = stLightCtr.iChannel2ActValue  // 通道2值匹配
    AND stLightCtr.iChannel3ValueSet = stLightCtr.iChannel3ActValue  // 通道3值匹配
    AND stLightCtr.iChannel4ValueSet = stLightCtr.iChannel4ActValue THEN  // 通道4值匹配
    // 所有值都匹配，无需更新
    bChanIntensityChgExe := FALSE;  // 设置亮度变化执行标志为FALSE（无需更新）
END_IF

//END_IF
//上升沿触发	 
// 配置200ms周期闪烁器（用于控制通信触发频率）
fbBlink1s(ENABLE := TRUE, TIMELOW := TIME#500MS, TIMEHIGH := TIME#500mS, OUT => );	 

// 检测亮度变化的上升沿（当变化标志从FALSE变为TRUE时触发）
rtrigChanIntensityChg(CLK := bChanIntensityChgExe AND fbBlink1s.OUT, Q => );	

// 如果检测到亮度变化的上升沿
IF rtrigChanIntensityChg.Q THEN
    iStep := 0;  // 重置状态机步骤为0（开始通信序列）
END_IF


// 配置步骤10的10ms超时定时器
Ton10(IN := iStep = 10, PT := TIME#10MS, Q => , ET => );
// 配置步骤20的20ms超时定时器
Ton20(IN := iStep = 20, PT := TIME#20MS, Q => , ET => );

// 状态机：控制通信流程的步骤
CASE iStep OF 
    0:  // 步骤0：初始化步骤
       iStep := 10;  // 直接跳转到步骤10（开始发送设置命令）
    
    10:  // 步骤10：发送设置命令
        // 调用发送功能块发送设置亮度数据帧
        fbSendData(
            pSendData := ADR(arSendData),           // 设置命令数据帧地址
            Length := SIZEOF(arSendData),           // 数据帧长度（字节数）
            Busy => ,                               // 输出：发送忙状态
            Error => ,                              // 输出：发送错误状态
            TXbuffer := TxBuffer_MASTER );          // 使用主站发送缓冲区
        
        // 如果10ms定时器到时且发送功能块不忙（发送完成）
        IF Ton10.Q AND NOT fbSendData.Busy THEN
          iStep := 20;  // 进入步骤20（发送读取命令）
        END_IF;        
        
    20:  // 步骤20：发送读取命令
        // 调用发送功能块发送读取亮度数据帧
        fbSendData2(
            pSendData := ADR(arSendData2),          // 读取命令数据帧地址
            Length := SIZEOF(arSendData2),          // 数据帧长度（字节数）
            Busy => ,                               // 输出：发送忙状态
            Error => ,                              // 输出：发送错误状态
            TXbuffer := TxBuffer_MASTER);           // 使用主站发送缓冲区
        
        // 如果20ms定时器到时且发送功能块不忙（发送完成）
        IF Ton20.Q AND NOT fbSendData2.Busy THEN
            iStep := 30;  // 进入步骤30（等待接收数据）
        END_IF;                
    30:
		 stLightCtr.iChannel1ActValue :=    (BYTE_TO_UINT(arReceiveData[5]));      // 或操作合并低字节
	 
       // 解析接收到的通道2亮度值
        stLightCtr.iChannel2ActValue :=  (BYTE_TO_UINT(arReceiveData[6]));      // 或操作合并低字节
	 
      // 解析接收到的通道3亮度值
      stLightCtr.iChannel3ActValue :=  (BYTE_TO_UINT(arReceiveData[7]));     // 或操作合并低字节
	 
     // 解析接收到的通道4亮度值
      stLightCtr.iChannel4ActValue := (BYTE_TO_UINT(arReceiveData[8]));     // 或操作合并低字节 
	  iStep:=40;
    // 步骤30：接收数据（隐含状态，由下面的接收功能块处理）
END_CASE

// 配置数据接收功能块（等待接收返回数据）
fbReceiveData(
    pPrefix := ADR(byStart),            // 数据帧前缀（起始字节0x40的地址）
    LenPrefix := 1,                     // 前缀长度（1字节）
    pSuffix := ,                        // 数据帧后缀
    LenSuffix := ,                      // 后缀长度
    pReceiveData := ADR(arReceiveData), // 接收数据缓冲区地址
    SizeReceiveData := SIZEOF(arReceiveData),  // 接收缓冲区大小
    Timeout := ,                        // 超时时间
    Reset := ,                          // 复位信号
    DataReceived => ,                   // 输出：数据接收完成标志
    busy => ,                           // 输出：接收忙状态
    Error => ,                          // 输出：接收错误状态
    RxTimeout => ,                      // 输出：接收超时标志
    LenReceiveData => ,                 // 输出：实际接收数据长度
    RXbuffer := RxBuffer_MASTER);       // 使用主站接收缓冲区

// 调用串口通信控制功能块（管理底层硬件通信）
fbSerialLineControl(
    Mode := SERIALLINEMODE_EL6_22B,     // 设置通信模式为EL6 22字节模式
    pComIn := ADR(COMin_MASTER),        // 输入缓冲区地址（硬件映射）
    pComOut := ADR(COMout_MASTER),      // 输出缓冲区地址（硬件映射）
    SizeComIn := UINT_TO_INT(SIZEOF(COMin_MASTER)),  // 输入缓冲区大小
    Error => ,                          // 输出：通信错误标志
    ErrorID => ,                        // 输出：错误代码
    TxBuffer := TxBuffer_MASTER,        // 发送缓冲区
    RxBuffer := RxBuffer_MASTER );      // 接收缓冲区

// 解析接收到的通道1亮度值（2个字节合并为16位整数）
//	 IF(iStep=30) THEN
//	   stLightCtr.iChannel1ActValue :=    (BYTE_TO_UINT(arReceiveData[5]));      // 或操作合并低字节
	 
//       // 解析接收到的通道2亮度值
//        stLightCtr.iChannel2ActValue :=  (BYTE_TO_UINT(arReceiveData[6]));      // 或操作合并低字节
	 
//      // 解析接收到的通道3亮度值
//      stLightCtr.iChannel3ActValue :=  (BYTE_TO_UINT(arReceiveData[7]));     // 或操作合并低字节
	 
//     // 解析接收到的通道4亮度值
//      stLightCtr.iChannel4ActValue := (BYTE_TO_UINT(arReceiveData[8]));     // 或操作合并低字节 
//  END_IF

END_FUNCTION_BLOCK

// ---- POUs/06_真空控制/Vac_Ctrl.TcPOU
PROGRAM Vac_Ctrl
VAR
    Vacuums     : ARRAY[1..4] OF ST_Vacuum;
    VacuumFB    : ARRAY[1..4] OF FB_VacuumControl;
    bResetAll   : BOOL;
    i           : INT;
END_VAR








(* 输出 *)
//Y000212 := stVac[1].qVacuumValve;
//Y000213 := stVac[1].qReleaseValve;
//Y000214 := stVac[2].qVacuumValve;
//Y000215 := stVac[2].qReleaseValve;

END_PROGRAM

// ---- FB/06真空控制/FB_VacuumControl.TcPOU
FUNCTION_BLOCK FB_VacuumControl


VAR_INPUT
    bVacuumReq      : BOOL;      // 抽真空请求
    bReleaseReq     : BOOL;      // 破真空请求
    bVacuumOk       : BOOL;      // 真空到位信号
    bResetAlarm     : BOOL;      // 报警复位
END_VAR

VAR_OUTPUT
    qVacuumValve    : BOOL;      // 真空阀输出
    qReleaseValve   : BOOL;      // 破真空阀输出
    bVacuumDone     : BOOL;      // 吸附完成
    bReleaseDone    : BOOL;      // 破真空完成
    bAlarm          : BOOL;      // 报警
END_VAR

VAR
    tVacuumTimer    : TON;       // 吸附超时定时器
    tReleaseTimer   : TON;       // 破真空定时器

    tMaxVacuumTime  : TIME := T#3S;      // 吸附超时
    tReleaseTime    : TIME := T#500MS;   // 破真空时间
END_VAR

// ===============================
// 1️⃣ 抽真空控制
// ===============================

qVacuumValve := bVacuumReq AND NOT bReleaseReq;

// 真空完成判断
bVacuumDone := bVacuumOk;


// 吸附超时检测
tVacuumTimer(
    IN := bVacuumReq AND NOT bVacuumOk,
    PT := tMaxVacuumTime
);

IF tVacuumTimer.Q THEN
    bAlarm := TRUE;
END_IF;


// ===============================
// 2️⃣ 破真空控制（定时自动关闭）
// ===============================
tReleaseTimer(
    IN := bReleaseReq,
    PT := tReleaseTime
);

// 破真空输出控制
qReleaseValve := bReleaseReq;


// 破真空完成判断
IF tReleaseTimer.Q THEN
    bReleaseDone := TRUE;
END_IF;


// 请求撤销自动复位完成信号
IF NOT bReleaseReq THEN
    bReleaseDone := FALSE;
END_IF;

// ===============================
// 3️⃣ 报警复位
// ===============================

IF bResetAlarm THEN
    bAlarm := FALSE;
END_IF;

END_FUNCTION_BLOCK

// ---- POUs/13_PosCompartion/POS_Comparition.TcPOU
PROGRAM POS_Comparition
VAR
	fbPOS_ComparitionXY:FB_013_POS_Comparition;
	fbPOS_ComparitionZR:FB_013_POS_Comparition;
END_VAR

// XY位置比较
fbPOS_ComparitionXY(arstCamCtrl:=arstCamCtrlIO, fbstIJP:=stIJP , stAxis:=arstAxis );

END_PROGRAM

